SPLINE
SPL {X  -160.000, Y  +472.196, Z    +0.000, E1   +56.977, E3 +201376.828}
SPL {X  -160.000, Y  +448.172, Z    +0.000, E1   +58.434, E3 +201399.523}
SPL {X  -160.000, Y  +423.986, Z    +0.000, E1   +59.836, E3 +201420.777}
SPL {X  -160.000, Y  +398.875, Z    +0.000, E1   +61.100, E3 +201442.325}
SPL {X  -159.733, Y  +376.466, Z    +0.000, E1   +61.765, E3 +201463.514}
SPL {X  -158.128, Y  +361.299, Z    +0.000, E1   +61.520, E3 +201482.494}
SPL {X  -155.661, Y  +348.690, Z    +0.000, E1   +61.132, E3 +201499.450}
SPL {X  -152.251, Y  +336.510, Z    +0.000, E1   +60.617, E3 +201516.783}
SPL {X  -148.078, Y  +325.096, Z    +0.000, E1   +59.928, E3 +201533.911}
SPL {X  -143.290, Y  +314.510, Z    +0.000, E1   +59.129, E3 +201550.534}
SPL {X  -139.113, Y  +306.659, Z    +0.000, E1   +58.310, E3 +201563.385}
SPL {X  -135.700, Y  +300.932, Z    +0.000, E1   +57.683, E3 +201572.881}
SPL {X  -117.539, Y  +277.143, Z    +0.000, E1   +48.559, E3 +201687.567}
ENDSPLINE

SPLINE
SPL {X  -150.734, Y  +332.041, Z    +0.000, E1   +31.286, E3 +201790.232}
SPL {X  -159.235, Y  +370.077, Z    +0.000, E1   +12.240, E3 +201803.586}
SPL {X  -159.991, Y  +384.025, Z    +0.000, E1    +2.884, E3 +201805.135}
SPL {X  -160.000, Y  +388.170, Z    +0.000, E1    -0.470, E3 +201805.266}
SPL {X  -160.000, Y  +392.385, Z    +0.000, E1    -5.697, E3 +201805.456}
SPL {X  -160.000, Y  +398.918, Z    +0.000, E1   -15.420, E3 +201806.134}
SPL {X  -160.000, Y  +410.991, Z    +0.000, E1   -32.499, E3 +201808.629}
SPL {X  -160.000, Y  +455.466, Z    +0.000, E1   -56.407, E3 +201829.528}
SPL {X  -160.000, Y  +554.875, Z    +0.000, E1   -61.915, E3 +201911.432}
SPL {X  -160.000, Y  +571.700, Z    +0.000, E1   -61.918, E3 +201930.509}
SPL {X  -160.000, Y  +587.975, Z    +0.000, E1   -61.909, E3 +201948.976}
SPL {X  -160.000, Y  +604.690, Z    +0.000, E1   -61.922, E3 +201967.905}
SPL {X  -160.000, Y  +621.475, Z    +0.000, E1   -61.913, E3 +201986.957}
SPL {X  -160.000, Y  +638.005, Z    +0.000, E1   -61.917, E3 +202005.687}
SPL {X  -160.000, Y  +655.083, Z    +0.000, E1   -61.921, E3 +202025.048}
SPL {X  -160.000, Y  +671.910, Z    +0.000, E1   -61.915, E3 +202044.142}
SPL {X  -159.476, Y  +687.338, Z    +0.000, E1   -61.835, E3 +202062.194}
SPL {X  -157.928, Y  +700.064, Z    +0.000, E1   -61.593, E3 +202078.259}
SPL {X  -155.236, Y  +713.154, Z    +0.000, E1   -61.225, E3 +202095.806}
SPL {X  -151.860, Y  +724.785, Z    +0.000, E1   -60.654, E3 +202112.479}
SPL {X  -148.451, Y  +734.085, Z    +0.000, E1   -60.099, E3 +202126.404}
SPL {X  -144.033, Y  +744.073, Z    +0.000, E1   -59.381, E3 +202141.924}
SPL {X  -139.170, Y  +753.341, Z    +0.000, E1   -58.489, E3 +202156.945}
SPL {X  -135.320, Y  +759.772, Z    +0.000, E1   -57.727, E3 +202167.655}
SPL {X  -117.185, Y  +783.339, Z    +0.000, E1   -48.966, E3 +202276.041}
ENDSPLINE

SPLINE
SPL {X  -142.074, Y  +747.987, Z    +0.000, E1   -38.326, E3 +202374.735}
SPL {X  -154.075, Y  +717.539, Z    +0.000, E1   -26.988, E3 +202393.892}
SPL {X  -158.904, Y  +693.092, Z    +0.000, E1   -14.171, E3 +202400.683}
SPL {X  -159.937, Y  +678.885, Z    +0.000, E1    -4.971, E3 +202402.510}
SPL {X  -160.000, Y  +672.790, Z    +0.000, E1    -0.387, E3 +202402.778}
SPL {X  -160.000, Y  +669.961, Z    +0.000, E1    +2.696, E3 +202402.855}
SPL {X  -160.000, Y  +663.591, Z    +0.000, E1   +11.688, E3 +202403.349}
SPL {X  -160.000, Y  +654.521, Z    +0.000, E1   +25.997, E3 +202404.707}
SPL {X  -160.000, Y  +642.364, Z    +0.000, E1   +40.387, E3 +202408.009}
SPL {X  -160.000, Y  +597.330, Z    +0.000, E1   +58.145, E3 +202430.920}
SPL {X  -160.000, Y  +516.293, Z    +0.000, E1   +61.751, E3 +202497.977}
SPL {X  -160.000, Y  +506.292, Z    +0.000, E1   +61.780, E3 +202509.311}
SPL {X  -160.000, Y  +494.139, Z    +0.000, E1   +61.770, E3 +202523.182}
SPL {X  -160.000, Y  +480.560, Z    +0.000, E1   +61.503, E3 +202540.979}
ENDSPLINE

SPLINE
SPL {X  -160.000, Y  +495.136, Z    +0.000, E1   +55.416, E3 +202562.485}
ENDSPLINE

SPLINE
SPL {X  -160.000, Y  +472.196, Z    +0.000, E1   +56.977, E3 +202585.160}
SPL {X  -160.000, Y  +448.172, Z    +0.000, E1   +58.434, E3 +202607.855}
SPL {X  -160.000, Y  +423.986, Z    +0.000, E1   +59.836, E3 +202629.108}
SPL {X  -160.000, Y  +398.875, Z    +0.000, E1   +61.100, E3 +202650.656}
SPL {X  -159.733, Y  +376.466, Z    +0.000, E1   +61.765, E3 +202671.846}
SPL {X  -158.128, Y  +361.299, Z    +0.000, E1   +61.520, E3 +202690.826}
SPL {X  -155.661, Y  +348.690, Z    +0.000, E1   +61.132, E3 +202707.782}
SPL {X  -152.251, Y  +336.510, Z    +0.000, E1   +60.617, E3 +202725.114}
SPL {X  -148.078, Y  +325.096, Z    +0.000, E1   +59.928, E3 +202742.243}
SPL {X  -143.290, Y  +314.510, Z    +0.000, E1   +59.129, E3 +202758.866}
SPL {X  -139.113, Y  +306.659, Z    +0.000, E1   +58.310, E3 +202771.716}
SPL {X  -135.700, Y  +300.932, Z    +0.000, E1   +57.683, E3 +202781.213}
SPL {X  -117.539, Y  +277.143, Z    +0.000, E1   +48.559, E3 +202895.899}
ENDSPLINE

SPLINE
SPL {X  -150.734, Y  +332.041, Z    +0.000, E1   +31.286, E3 +202998.564}
SPL {X  -159.235, Y  +370.077, Z    +0.000, E1   +12.240, E3 +203011.918}
SPL {X  -159.991, Y  +384.025, Z    +0.000, E1    +2.884, E3 +203013.467}
SPL {X  -160.000, Y  +388.170, Z    +0.000, E1    -0.470, E3 +203013.597}
SPL {X  -160.000, Y  +392.385, Z    +0.000, E1    -5.697, E3 +203013.787}
SPL {X  -160.000, Y  +398.918, Z    +0.000, E1   -15.420, E3 +203014.466}
SPL {X  -160.000, Y  +410.991, Z    +0.000, E1   -32.499, E3 +203016.961}
SPL {X  -160.000, Y  +455.466, Z    +0.000, E1   -56.407, E3 +203037.860}
SPL {X  -160.000, Y  +554.875, Z    +0.000, E1   -61.915, E3 +203119.764}
SPL {X  -160.000, Y  +571.700, Z    +0.000, E1   -61.918, E3 +203138.841}
SPL {X  -160.000, Y  +587.975, Z    +0.000, E1   -61.909, E3 +203157.307}
SPL {X  -160.000, Y  +604.690, Z    +0.000, E1   -61.922, E3 +203176.237}
SPL {X  -160.000, Y  +621.475, Z    +0.000, E1   -61.913, E3 +203195.288}
SPL {X  -160.000, Y  +638.005, Z    +0.000, E1   -61.917, E3 +203214.019}
SPL {X  -160.000, Y  +655.083, Z    +0.000, E1   -61.921, E3 +203233.380}
SPL {X  -160.000, Y  +671.910, Z    +0.000, E1   -61.915, E3 +203252.474}
SPL {X  -159.476, Y  +687.338, Z    +0.000, E1   -61.835, E3 +203270.526}
SPL {X  -157.928, Y  +700.064, Z    +0.000, E1   -61.593, E3 +203286.591}
SPL {X  -155.236, Y  +713.154, Z    +0.000, E1   -61.225, E3 +203304.138}
SPL {X  -151.860, Y  +724.785, Z    +0.000, E1   -60.654, E3 +203320.810}
SPL {X  -148.451, Y  +734.085, Z    +0.000, E1   -60.099, E3 +203334.735}
SPL {X  -144.033, Y  +744.073, Z    +0.000, E1   -59.381, E3 +203350.256}
SPL {X  -139.170, Y  +753.341, Z    +0.000, E1   -58.489, E3 +203365.277}
SPL {X  -135.320, Y  +759.772, Z    +0.000, E1   -57.727, E3 +203375.987}
SPL {X  -117.185, Y  +783.339, Z    +0.000, E1   -48.966, E3 +203484.373}
ENDSPLINE

SPLINE
SPL {X  -142.074, Y  +747.987, Z    +0.000, E1   -38.326, E3 +203583.067}
SPL {X  -154.075, Y  +717.539, Z    +0.000, E1   -26.988, E3 +203602.224}
SPL {X  -158.904, Y  +693.092, Z    +0.000, E1   -14.171, E3 +203609.015}
SPL {X  -159.937, Y  +678.885, Z    +0.000, E1    -4.971, E3 +203610.842}
SPL {X  -160.000, Y  +672.790, Z    +0.000, E1    -0.387, E3 +203611.110}
SPL {X  -160.000, Y  +669.961, Z    +0.000, E1    +2.696, E3 +203611.187}
SPL {X  -160.000, Y  +663.591, Z    +0.000, E1   +11.688, E3 +203611.681}
SPL {X  -160.000, Y  +654.521, Z    +0.000, E1   +25.997, E3 +203613.039}
SPL {X  -160.000, Y  +642.364, Z    +0.000, E1   +40.387, E3 +203616.341}
SPL {X  -160.000, Y  +597.330, Z    +0.000, E1   +58.145, E3 +203639.252}
SPL {X  -160.000, Y  +507.195, Z    +0.000, E1   +61.792, E3 +203716.583}
SPL {X  -160.000, Y  +494.139, Z    +0.000, E1   +61.770, E3 +203731.513}
SPL {X  -160.000, Y  +480.560, Z    +0.000, E1   +61.503, E3 +203749.310}
ENDSPLINE

SPLINE
SPL {X  -160.000, Y  +495.136, Z    +0.000, E1   +55.416, E3 +203770.817}
ENDSPLINE

SPLINE
SPL {X  -160.000, Y  +472.196, Z    +0.000, E1   +56.977, E3 +203793.492}
SPL {X  -160.000, Y  +448.172, Z    +0.000, E1   +58.434, E3 +203816.187}
SPL {X  -160.000, Y  +423.986, Z    +0.000, E1   +59.836, E3 +203837.440}
SPL {X  -160.000, Y  +398.875, Z    +0.000, E1   +61.100, E3 +203858.988}
SPL {X  -159.733, Y  +376.466, Z    +0.000, E1   +61.765, E3 +203880.178}
SPL {X  -158.128, Y  +361.299, Z    +0.000, E1   +61.520, E3 +203899.157}
SPL {X  -155.661, Y  +348.690, Z    +0.000, E1   +61.132, E3 +203916.113}
SPL {X  -152.251, Y  +336.510, Z    +0.000, E1   +60.617, E3 +203933.446}
SPL {X  -148.078, Y  +325.096, Z    +0.000, E1   +59.928, E3 +203950.575}
SPL {X  -143.290, Y  +314.510, Z    +0.000, E1   +59.129, E3 +203967.198}
SPL {X  -139.113, Y  +306.659, Z    +0.000, E1   +58.310, E3 +203980.048}
SPL {X  -135.700, Y  +300.932, Z    +0.000, E1   +57.683, E3 +203989.545}
SPL {X  -117.539, Y  +277.143, Z    +0.000, E1   +48.559, E3 +204104.231}
ENDSPLINE

SPLINE
SPL {X  -150.734, Y  +332.041, Z    +0.000, E1   +31.286, E3 +204206.896}
SPL {X  -159.235, Y  +370.077, Z    +0.000, E1   +12.240, E3 +204220.250}
SPL {X  -159.991, Y  +384.025, Z    +0.000, E1    +2.884, E3 +204221.798}
SPL {X  -160.000, Y  +388.170, Z    +0.000, E1    -0.470, E3 +204221.929}
SPL {X  -160.000, Y  +392.385, Z    +0.000, E1    -5.697, E3 +204222.119}
SPL {X  -160.000, Y  +398.918, Z    +0.000, E1   -15.420, E3 +204222.798}
SPL {X  -160.000, Y  +410.991, Z    +0.000, E1   -32.499, E3 +204225.293}
SPL {X  -160.000, Y  +455.466, Z    +0.000, E1   -56.407, E3 +204246.192}
SPL {X  -160.000, Y  +554.875, Z    +0.000, E1   -61.915, E3 +204328.096}
SPL {X  -160.000, Y  +571.700, Z    +0.000, E1   -61.918, E3 +204347.173}
SPL {X  -160.000, Y  +587.975, Z    +0.000, E1   -61.909, E3 +204365.639}
SPL {X  -160.000, Y  +604.690, Z    +0.000, E1   -61.922, E3 +204384.568}
SPL {X  -160.000, Y  +621.475, Z    +0.000, E1   -61.913, E3 +204403.620}
SPL {X  -160.000, Y  +638.005, Z    +0.000, E1   -61.917, E3 +204422.351}
SPL {X  -160.000, Y  +655.083, Z    +0.000, E1   -61.921, E3 +204441.712}
SPL {X  -160.000, Y  +671.910, Z    +0.000, E1   -61.915, E3 +204460.806}
SPL {X  -159.476, Y  +687.338, Z    +0.000, E1   -61.835, E3 +204478.858}
SPL {X  -157.928, Y  +700.064, Z    +0.000, E1   -61.593, E3 +204494.922}
SPL {X  -155.236, Y  +713.154, Z    +0.000, E1   -61.225, E3 +204512.469}
SPL {X  -151.860, Y  +724.785, Z    +0.000, E1   -60.654, E3 +204529.142}
SPL {X  -148.451, Y  +734.085, Z    +0.000, E1   -60.099, E3 +204543.067}
SPL {X  -144.033, Y  +744.073, Z    +0.000, E1   -59.381, E3 +204558.587}
SPL {X  -139.170, Y  +753.341, Z    +0.000, E1   -58.489, E3 +204573.609}
SPL {X  -135.320, Y  +759.772, Z    +0.000, E1   -57.727, E3 +204584.319}
SPL {X  -117.185, Y  +783.339, Z    +0.000, E1   -48.966, E3 +204692.705}
ENDSPLINE

SPLINE
SPL {X  -142.074, Y  +747.987, Z    +0.000, E1   -38.326, E3 +204791.398}
SPL {X  -154.075, Y  +717.539, Z    +0.000, E1   -26.988, E3 +204810.555}
SPL {X  -158.904, Y  +693.092, Z    +0.000, E1   -14.171, E3 +204817.346}
SPL {X  -159.937, Y  +678.885, Z    +0.000, E1    -4.971, E3 +204819.174}
SPL {X  -160.000, Y  +672.790, Z    +0.000, E1    -0.387, E3 +204819.442}
SPL {X  -160.000, Y  +669.961, Z    +0.000, E1    +2.696, E3 +204819.518}
SPL {X  -160.000, Y  +663.591, Z    +0.000, E1   +11.688, E3 +204820.013}
SPL {X  -160.000, Y  +654.521, Z    +0.000, E1   +25.997, E3 +204821.370}
SPL {X  -160.000, Y  +642.364, Z    +0.000, E1   +40.387, E3 +204824.673}
SPL {X  -160.000, Y  +597.330, Z    +0.000, E1   +58.145, E3 +204847.584}
SPL {X  -160.000, Y  +507.195, Z    +0.000, E1   +61.792, E3 +204924.915}
SPL {X  -160.000, Y  +494.139, Z    +0.000, E1   +61.770, E3 +204939.845}
SPL {X  -160.000, Y  +480.560, Z    +0.000, E1   +61.503, E3 +204957.642}
ENDSPLINE

SPLINE
SPL {X  -160.000, Y  +495.136, Z    +0.000, E1   +55.416, E3 +204979.149}
ENDSPLINE

SPLINE
SPL {X  -160.000, Y  +472.196, Z    +0.000, E1   +56.977, E3 +205001.824}
SPL {X  -160.000, Y  +448.172, Z    +0.000, E1   +58.434, E3 +205024.518}
SPL {X  -160.000, Y  +423.986, Z    +0.000, E1   +59.836, E3 +205045.772}
SPL {X  -160.000, Y  +398.875, Z    +0.000, E1   +61.100, E3 +205067.320}
SPL {X  -159.733, Y  +376.466, Z    +0.000, E1   +61.765, E3 +205088.509}
SPL {X  -158.128, Y  +361.299, Z    +0.000, E1   +61.520, E3 +205107.489}
SPL {X  -155.661, Y  +348.690, Z    +0.000, E1   +61.132, E3 +205124.445}
SPL {X  -152.251, Y  +336.510, Z    +0.000, E1   +60.617, E3 +205141.778}
SPL {X  -148.078, Y  +325.096, Z    +0.000, E1   +59.928, E3 +205158.906}
SPL {X  -143.290, Y  +314.510, Z    +0.000, E1   +59.129, E3 +205175.529}
SPL {X  -139.113, Y  +306.659, Z    +0.000, E1   +58.310, E3 +205188.380}
SPL {X  -135.700, Y  +300.932, Z    +0.000, E1   +57.683, E3 +205197.877}
SPL {X  -117.539, Y  +277.143, Z    +0.000, E1   +48.559, E3 +205312.563}
ENDSPLINE

SPLINE
SPL {X  -150.734, Y  +332.041, Z    +0.000, E1   +31.286, E3 +205415.227}
SPL {X  -159.235, Y  +370.077, Z    +0.000, E1   +12.240, E3 +205428.581}
SPL {X  -159.991, Y  +384.025, Z    +0.000, E1    +2.884, E3 +205430.130}
SPL {X  -160.000, Y  +388.170, Z    +0.000, E1    -0.470, E3 +205430.261}
SPL {X  -160.000, Y  +392.385, Z    +0.000, E1    -5.697, E3 +205430.451}
SPL {X  -160.000, Y  +398.918, Z    +0.000, E1   -15.420, E3 +205431.130}
SPL {X  -160.000, Y  +410.991, Z    +0.000, E1   -32.499, E3 +205433.625}
SPL {X  -160.000, Y  +455.466, Z    +0.000, E1   -56.407, E3 +205454.524}
SPL {X  -160.000, Y  +554.875, Z    +0.000, E1   -61.915, E3 +205536.427}
SPL {X  -160.000, Y  +571.700, Z    +0.000, E1   -61.918, E3 +205555.504}
SPL {X  -160.000, Y  +587.975, Z    +0.000, E1   -61.909, E3 +205573.971}
SPL {X  -160.000, Y  +604.690, Z    +0.000, E1   -61.922, E3 +205592.900}
SPL {X  -160.000, Y  +621.475, Z    +0.000, E1   -61.913, E3 +205611.952}
SPL {X  -160.000, Y  +638.005, Z    +0.000, E1   -61.917, E3 +205630.682}
SPL {X  -160.000, Y  +655.083, Z    +0.000, E1   -61.921, E3 +205650.044}
SPL {X  -160.000, Y  +671.910, Z    +0.000, E1   -61.915, E3 +205669.138}
SPL {X  -159.476, Y  +687.338, Z    +0.000, E1   -61.835, E3 +205687.190}
SPL {X  -157.928, Y  +700.064, Z    +0.000, E1   -61.593, E3 +205703.254}
SPL {X  -155.236, Y  +713.154, Z    +0.000, E1   -61.225, E3 +205720.801}
SPL {X  -151.860, Y  +724.785, Z    +0.000, E1   -60.654, E3 +205737.474}
SPL {X  -148.451, Y  +734.085, Z    +0.000, E1   -60.099, E3 +205751.399}
SPL {X  -144.033, Y  +744.073, Z    +0.000, E1   -59.381, E3 +205766.919}
SPL {X  -139.170, Y  +753.341, Z    +0.000, E1   -58.489, E3 +205781.941}
SPL {X  -135.320, Y  +759.772, Z    +0.000, E1   -57.727, E3 +205792.650}
SPL {X  -117.185, Y  +783.339, Z    +0.000, E1   -48.966, E3 +205901.037}
ENDSPLINE

SPLINE
SPL {X  -142.074, Y  +747.987, Z    +0.000, E1   -38.326, E3 +205999.730}
SPL {X  -154.075, Y  +717.539, Z    +0.000, E1   -26.988, E3 +206018.887}
SPL {X  -158.904, Y  +693.092, Z    +0.000, E1   -14.171, E3 +206025.678}
SPL {X  -159.937, Y  +678.885, Z    +0.000, E1    -4.971, E3 +206027.505}
SPL {X  -160.000, Y  +672.790, Z    +0.000, E1    -0.387, E3 +206027.773}
SPL {X  -160.000, Y  +669.961, Z    +0.000, E1    +2.696, E3 +206027.850}
SPL {X  -160.000, Y  +663.591, Z    +0.000, E1   +11.688, E3 +206028.344}
SPL {X  -160.000, Y  +654.521, Z    +0.000, E1   +25.997, E3 +206029.702}
SPL {X  -160.000, Y  +642.364, Z    +0.000, E1   +40.387, E3 +206033.004}
SPL {X  -160.000, Y  +597.330, Z    +0.000, E1   +58.145, E3 +206055.915}
SPL {X  -160.000, Y  +516.293, Z    +0.000, E1   +61.751, E3 +206122.973}
SPL {X  -160.000, Y  +506.292, Z    +0.000, E1   +61.780, E3 +206134.306}
SPL {X  -160.000, Y  +494.139, Z    +0.000, E1   +61.770, E3 +206148.177}
SPL {X  -160.000, Y  +480.560, Z    +0.000, E1   +61.503, E3 +206165.974}
ENDSPLINE

SPLINE
SPL {X  -160.000, Y  +495.136, Z    +0.000, E1   +55.416, E3 +206187.480}
ENDSPLINE

SPLINE
SPL {X  -160.000, Y  +472.196, Z    +0.000, E1   +56.977, E3 +206210.155}
SPL {X  -160.000, Y  +448.172, Z    +0.000, E1   +58.434, E3 +206232.850}
SPL {X  -160.000, Y  +423.986, Z    +0.000, E1   +59.836, E3 +206254.104}
SPL {X  -160.000, Y  +398.875, Z    +0.000, E1   +61.100, E3 +206275.652}
SPL {X  -159.733, Y  +376.466, Z    +0.000, E1   +61.765, E3 +206296.841}
SPL {X  -158.128, Y  +361.299, Z    +0.000, E1   +61.520, E3 +206315.821}
SPL {X  -155.661, Y  +348.690, Z    +0.000, E1   +61.132, E3 +206332.777}
SPL {X  -152.251, Y  +336.510, Z    +0.000, E1   +60.617, E3 +206350.110}
SPL {X  -148.078, Y  +325.096, Z    +0.000, E1   +59.928, E3 +206367.238}
SPL {X  -143.290, Y  +314.510, Z    +0.000, E1   +59.129, E3 +206383.861}
SPL {X  -139.113, Y  +306.659, Z    +0.000, E1   +58.310, E3 +206396.712}
SPL {X  -135.700, Y  +300.932, Z    +0.000, E1   +57.683, E3 +206406.208}
SPL {X  -117.539, Y  +277.143, Z    +0.000, E1   +48.559, E3 +206520.894}
ENDSPLINE

SPLINE
SPL {X  -150.734, Y  +332.041, Z    +0.000, E1   +31.286, E3 +206623.559}
SPL {X  -159.235, Y  +370.077, Z    +0.000, E1   +12.240, E3 +206636.913}
SPL {X  -159.991, Y  +384.025, Z    +0.000, E1    +2.884, E3 +206638.462}
SPL {X  -160.000, Y  +388.170, Z    +0.000, E1    -0.470, E3 +206638.593}
SPL {X  -160.000, Y  +392.385, Z    +0.000, E1    -5.697, E3 +206638.783}
SPL {X  -160.000, Y  +398.918, Z    +0.000, E1   -15.420, E3 +206639.461}
SPL {X  -160.000, Y  +410.991, Z    +0.000, E1   -32.499, E3 +206641.956}
SPL {X  -160.000, Y  +455.466, Z    +0.000, E1   -56.407, E3 +206662.855}
SPL {X  -160.000, Y  +554.875, Z    +0.000, E1   -61.915, E3 +206744.759}
SPL {X  -160.000, Y  +571.700, Z    +0.000, E1   -61.918, E3 +206763.836}
SPL {X  -160.000, Y  +587.975, Z    +0.000, E1   -61.909, E3 +206782.303}
SPL {X  -160.000, Y  +604.690, Z    +0.000, E1   -61.922, E3 +206801.232}
SPL {X  -160.000, Y  +621.475, Z    +0.000, E1   -61.913, E3 +206820.284}
SPL {X  -160.000, Y  +638.005, Z    +0.000, E1   -61.917, E3 +206839.014}
SPL {X  -160.000, Y  +655.083, Z    +0.000, E1   -61.921, E3 +206858.375}
SPL {X  -160.000, Y  +671.910, Z    +0.000, E1   -61.915, E3 +206877.469}
SPL {X  -159.476, Y  +687.338, Z    +0.000, E1   -61.835, E3 +206895.521}
SPL {X  -157.928, Y  +700.064, Z    +0.000, E1   -61.593, E3 +206911.586}
SPL {X  -155.236, Y  +713.154, Z    +0.000, E1   -61.225, E3 +206929.133}
SPL {X  -151.860, Y  +724.785, Z    +0.000, E1   -60.654, E3 +206945.806}
SPL {X  -148.451, Y  +734.085, Z    +0.000, E1   -60.099, E3 +206959.731}
SPL {X  -144.033, Y  +744.073, Z    +0.000, E1   -59.381, E3 +206975.251}
SPL {X  -139.170, Y  +753.341, Z    +0.000, E1   -58.489, E3 +206990.273}
SPL {X  -135.320, Y  +759.772, Z    +0.000, E1   -57.727, E3 +207000.982}
SPL {X  -117.185, Y  +783.339, Z    +0.000, E1   -48.966, E3 +207109.368}
ENDSPLINE

SPLINE
SPL {X  -142.074, Y  +747.987, Z    +0.000, E1   -38.326, E3 +207208.062}
SPL {X  -154.075, Y  +717.539, Z    +0.000, E1   -26.988, E3 +207227.219}
SPL {X  -158.904, Y  +693.092, Z    +0.000, E1   -14.171, E3 +207234.010}
SPL {X  -159.937, Y  +678.885, Z    +0.000, E1    -4.971, E3 +207235.837}
SPL {X  -160.000, Y  +672.790, Z    +0.000, E1    -0.387, E3 +207236.105}
SPL {X  -160.000, Y  +669.961, Z    +0.000, E1    +2.696, E3 +207236.182}
SPL {X  -160.000, Y  +663.591, Z    +0.000, E1   +11.688, E3 +207236.676}
SPL {X  -160.000, Y  +654.521, Z    +0.000, E1   +25.997, E3 +207238.034}
SPL {X  -160.000, Y  +642.364, Z    +0.000, E1   +40.387, E3 +207241.336}
SPL {X  -160.000, Y  +597.330, Z    +0.000, E1   +58.145, E3 +207264.247}
SPL {X  -160.000, Y  +507.195, Z    +0.000, E1   +61.792, E3 +207341.578}
SPL {X  -160.000, Y  +494.139, Z    +0.000, E1   +61.770, E3 +207356.509}
SPL {X  -160.000, Y  +480.560, Z    +0.000, E1   +61.503, E3 +207374.306}
ENDSPLINE

SPLINE
SPL {X  -160.000, Y  +495.136, Z    +0.000, E1   +55.416, E3 +207395.812}
ENDSPLINE

SPLINE
SPL {X  -160.000, Y  +472.196, Z    +0.000, E1   +56.977, E3 +207418.487}
SPL {X  -160.000, Y  +448.172, Z    +0.000, E1   +58.434, E3 +207441.182}
SPL {X  -160.000, Y  +423.986, Z    +0.000, E1   +59.836, E3 +207462.435}
SPL {X  -160.000, Y  +398.875, Z    +0.000, E1   +61.100, E3 +207483.983}
SPL {X  -159.733, Y  +376.466, Z    +0.000, E1   +61.765, E3 +207505.173}
SPL {X  -158.128, Y  +361.299, Z    +0.000, E1   +61.520, E3 +207524.153}
SPL {X  -155.661, Y  +348.690, Z    +0.000, E1   +61.132, E3 +207541.109}
SPL {X  -152.251, Y  +336.510, Z    +0.000, E1   +60.617, E3 +207558.441}
SPL {X  -148.078, Y  +325.096, Z    +0.000, E1   +59.928, E3 +207575.570}
SPL {X  -143.290, Y  +314.510, Z    +0.000, E1   +59.129, E3 +207592.193}
SPL {X  -139.113, Y  +306.659, Z    +0.000, E1   +58.310, E3 +207605.043}
SPL {X  -135.700, Y  +300.932, Z    +0.000, E1   +57.683, E3 +207614.540}
SPL {X  -117.539, Y  +277.143, Z    +0.000, E1   +48.559, E3 +207729.226}
ENDSPLINE

SPLINE
SPL {X  -150.734, Y  +332.041, Z    +0.000, E1   +31.286, E3 +207831.891}
SPL {X  -159.235, Y  +370.077, Z    +0.000, E1   +12.240, E3 +207845.245}
SPL {X  -159.991, Y  +384.025, Z    +0.000, E1    +2.884, E3 +207846.794}
SPL {X  -160.000, Y  +388.170, Z    +0.000, E1    -0.470, E3 +207846.924}
SPL {X  -160.000, Y  +392.385, Z    +0.000, E1    -5.697, E3 +207847.114}
SPL {X  -160.000, Y  +398.918, Z    +0.000, E1   -15.420, E3 +207847.793}
SPL {X  -160.000, Y  +410.991, Z    +0.000, E1   -32.499, E3 +207850.288}
SPL {X  -160.000, Y  +455.466, Z    +0.000, E1   -56.407, E3 +207871.187}
SPL {X  -160.000, Y  +554.875, Z    +0.000, E1   -61.915, E3 +207953.091}
SPL {X  -160.000, Y  +571.700, Z    +0.000, E1   -61.918, E3 +207972.168}
SPL {X  -160.000, Y  +587.975, Z    +0.000, E1   -61.909, E3 +207990.634}
SPL {X  -160.000, Y  +604.690, Z    +0.000, E1   -61.922, E3 +208009.564}
SPL {X  -160.000, Y  +621.475, Z    +0.000, E1   -61.913, E3 +208028.615}
SPL {X  -160.000, Y  +638.005, Z    +0.000, E1   -61.917, E3 +208047.346}
SPL {X  -160.000, Y  +655.083, Z    +0.000, E1   -61.921, E3 +208066.707}
SPL {X  -160.000, Y  +671.910, Z    +0.000, E1   -61.915, E3 +208085.801}
SPL {X  -159.476, Y  +687.338, Z    +0.000, E1   -61.835, E3 +208103.853}
SPL {X  -157.928, Y  +700.064, Z    +0.000, E1   -61.593, E3 +208119.918}
SPL {X  -155.236, Y  +713.154, Z    +0.000, E1   -61.225, E3 +208137.465}
SPL {X  -151.860, Y  +724.785, Z    +0.000, E1   -60.654, E3 +208154.137}
SPL {X  -148.451, Y  +734.085, Z    +0.000, E1   -60.099, E3 +208168.062}
SPL {X  -144.033, Y  +744.073, Z    +0.000, E1   -59.381, E3 +208183.583}
SPL {X  -139.170, Y  +753.341, Z    +0.000, E1   -58.489, E3 +208198.604}
SPL {X  -135.320, Y  +759.772, Z    +0.000, E1   -57.727, E3 +208209.314}
SPL {X  -117.185, Y  +783.339, Z    +0.000, E1   -48.966, E3 +208317.700}
ENDSPLINE

SPLINE
SPL {X  -142.074, Y  +747.987, Z    +0.000, E1   -38.326, E3 +208416.394}
SPL {X  -154.075, Y  +717.539, Z    +0.000, E1   -26.988, E3 +208435.551}
SPL {X  -158.904, Y  +693.092, Z    +0.000, E1   -14.171, E3 +208442.342}
SPL {X  -159.937, Y  +678.885, Z    +0.000, E1    -4.971, E3 +208444.169}
SPL {X  -160.000, Y  +672.790, Z    +0.000, E1    -0.387, E3 +208444.437}
SPL {X  -160.000, Y  +669.961, Z    +0.000, E1    +2.696, E3 +208444.514}
SPL {X  -160.000, Y  +663.591, Z    +0.000, E1   +11.688, E3 +208445.008}
SPL {X  -160.000, Y  +654.521, Z    +0.000, E1   +25.997, E3 +208446.366}
SPL {X  -160.000, Y  +642.364, Z    +0.000, E1   +40.387, E3 +208449.668}
SPL {X  -160.000, Y  +597.330, Z    +0.000, E1   +58.145, E3 +208472.579}
SPL {X  -160.000, Y  +507.195, Z    +0.000, E1   +61.792, E3 +208549.910}
SPL {X  -160.000, Y  +494.139, Z    +0.000, E1   +61.770, E3 +208564.840}
SPL {X  -160.000, Y  +480.560, Z    +0.000, E1   +61.503, E3 +208582.637}
ENDSPLINE

SPLINE
SPL {X  -160.000, Y  +495.136, Z    +0.000, E1   +55.416, E3 +208604.144}
ENDSPLINE

SPLINE
SPL {X  -160.000, Y  +472.196, Z    +0.000, E1   +56.977, E3 +208626.819}
SPL {X  -160.000, Y  +448.172, Z    +0.000, E1   +58.434, E3 +208649.514}
SPL {X  -160.000, Y  +423.986, Z    +0.000, E1   +59.836, E3 +208670.767}
SPL {X  -160.000, Y  +398.875, Z    +0.000, E1   +61.100, E3 +208692.315}
SPL {X  -159.733, Y  +376.466, Z    +0.000, E1   +61.765, E3 +208713.505}
SPL {X  -158.128, Y  +361.299, Z    +0.000, E1   +61.520, E3 +208732.484}
SPL {X  -155.661, Y  +348.690, Z    +0.000, E1   +61.132, E3 +208749.440}
SPL {X  -152.251, Y  +336.510, Z    +0.000, E1   +60.617, E3 +208766.773}
SPL {X  -148.078, Y  +325.096, Z    +0.000, E1   +59.928, E3 +208783.902}
SPL {X  -143.290, Y  +314.510, Z    +0.000, E1   +59.129, E3 +208800.525}
SPL {X  -139.113, Y  +306.659, Z    +0.000, E1   +58.310, E3 +208813.375}
SPL {X  -135.700, Y  +300.932, Z    +0.000, E1   +57.683, E3 +208822.872}
SPL {X  -117.539, Y  +277.143, Z    +0.000, E1   +48.559, E3 +208937.558}
ENDSPLINE

SPLINE
SPL {X  -150.734, Y  +332.041, Z    +0.000, E1   +31.286, E3 +209040.223}
SPL {X  -159.235, Y  +370.077, Z    +0.000, E1   +12.240, E3 +209053.577}
SPL {X  -159.991, Y  +384.025, Z    +0.000, E1    +2.884, E3 +209055.125}
SPL {X  -160.000, Y  +388.170, Z    +0.000, E1    -0.470, E3 +209055.256}
SPL {X  -160.000, Y  +392.385, Z    +0.000, E1    -5.697, E3 +209055.446}
SPL {X  -160.000, Y  +398.918, Z    +0.000, E1   -15.420, E3 +209056.125}
SPL {X  -160.000, Y  +410.991, Z    +0.000, E1   -32.499, E3 +209058.620}
SPL {X  -160.000, Y  +455.466, Z    +0.000, E1   -56.407, E3 +209079.519}
SPL {X  -160.000, Y  +554.875, Z    +0.000, E1   -61.915, E3 +209161.423}
SPL {X  -160.000, Y  +571.700, Z    +0.000, E1   -61.918, E3 +209180.500}
SPL {X  -160.000, Y  +587.975, Z    +0.000, E1   -61.909, E3 +209198.966}
SPL {X  -160.000, Y  +604.690, Z    +0.000, E1   -61.922, E3 +209217.895}
SPL {X  -160.000, Y  +621.475, Z    +0.000, E1   -61.913, E3 +209236.947}
SPL {X  -160.000, Y  +638.005, Z    +0.000, E1   -61.917, E3 +209255.678}
SPL {X  -160.000, Y  +655.083, Z    +0.000, E1   -61.921, E3 +209275.039}
SPL {X  -160.000, Y  +671.910, Z    +0.000, E1   -61.915, E3 +209294.133}
SPL {X  -159.476, Y  +687.338, Z    +0.000, E1   -61.835, E3 +209312.185}
SPL {X  -157.928, Y  +700.064, Z    +0.000, E1   -61.593, E3 +209328.249}
SPL {X  -155.236, Y  +713.154, Z    +0.000, E1   -61.225, E3 +209345.797}
SPL {X  -151.860, Y  +724.785, Z    +0.000, E1   -60.654, E3 +209362.469}
SPL {X  -148.451, Y  +734.085, Z    +0.000, E1   -60.099, E3 +209376.394}
SPL {X  -144.033, Y  +744.073, Z    +0.000, E1   -59.381, E3 +209391.914}
SPL {X  -139.170, Y  +753.341, Z    +0.000, E1   -58.489, E3 +209406.936}
SPL {X  -135.320, Y  +759.772, Z    +0.000, E1   -57.727, E3 +209417.646}
SPL {X  -117.185, Y  +783.339, Z    +0.000, E1   -48.966, E3 +209526.032}
ENDSPLINE

SPLINE
SPL {X  -142.074, Y  +747.987, Z    +0.000, E1   -38.326, E3 +209624.725}
SPL {X  -154.075, Y  +717.539, Z    +0.000, E1   -26.988, E3 +209643.882}
SPL {X  -158.904, Y  +693.092, Z    +0.000, E1   -14.171, E3 +209650.673}
SPL {X  -159.937, Y  +678.885, Z    +0.000, E1    -4.971, E3 +209652.501}
SPL {X  -160.000, Y  +672.790, Z    +0.000, E1    -0.387, E3 +209652.769}
SPL {X  -160.000, Y  +669.961, Z    +0.000, E1    +2.696, E3 +209652.845}
SPL {X  -160.000, Y  +663.591, Z    +0.000, E1   +11.688, E3 +209653.340}
SPL {X  -160.000, Y  +654.521, Z    +0.000, E1   +25.997, E3 +209654.698}
SPL {X  -160.000, Y  +642.364, Z    +0.000, E1   +40.387, E3 +209658.000}
SPL {X  -160.000, Y  +597.330, Z    +0.000, E1   +58.145, E3 +209680.911}
SPL {X  -160.000, Y  +507.195, Z    +0.000, E1   +61.792, E3 +209758.242}
SPL {X  -160.000, Y  +494.139, Z    +0.000, E1   +61.770, E3 +209773.172}
SPL {X  -160.000, Y  +480.560, Z    +0.000, E1   +61.503, E3 +209790.969}
ENDSPLINE

SPLINE
SPL {X  -160.000, Y  +495.136, Z    +0.000, E1   +55.416, E3 +209812.476}
ENDSPLINE

SPLINE
SPL {X  -160.000, Y  +472.196, Z    +0.000, E1   +56.977, E3 +209835.151}
SPL {X  -160.000, Y  +448.172, Z    +0.000, E1   +58.434, E3 +209857.845}
SPL {X  -160.000, Y  +423.986, Z    +0.000, E1   +59.836, E3 +209879.099}
SPL {X  -160.000, Y  +398.875, Z    +0.000, E1   +61.100, E3 +209900.647}
SPL {X  -159.733, Y  +376.466, Z    +0.000, E1   +61.765, E3 +209921.837}
SPL {X  -158.128, Y  +361.299, Z    +0.000, E1   +61.520, E3 +209940.816}
SPL {X  -155.661, Y  +348.690, Z    +0.000, E1   +61.132, E3 +209957.772}
SPL {X  -152.251, Y  +336.510, Z    +0.000, E1   +60.617, E3 +209975.105}
SPL {X  -148.078, Y  +325.096, Z    +0.000, E1   +59.928, E3 +209992.233}
SPL {X  -143.290, Y  +314.510, Z    +0.000, E1   +59.129, E3 +210008.856}
SPL {X  -139.113, Y  +306.659, Z    +0.000, E1   +58.310, E3 +210021.707}
SPL {X  -135.700, Y  +300.932, Z    +0.000, E1   +57.683, E3 +210031.204}
SPL {X  -117.539, Y  +277.143, Z    +0.000, E1   +48.559, E3 +210145.890}
ENDSPLINE

SPLINE
SPL {X  -150.734, Y  +332.041, Z    +0.000, E1   +31.286, E3 +210248.554}
SPL {X  -159.235, Y  +370.077, Z    +0.000, E1   +12.240, E3 +210261.909}
SPL {X  -159.991, Y  +384.025, Z    +0.000, E1    +2.884, E3 +210263.457}
SPL {X  -160.000, Y  +388.170, Z    +0.000, E1    -0.470, E3 +210263.588}
SPL {X  -160.000, Y  +392.385, Z    +0.000, E1    -5.697, E3 +210263.778}
SPL {X  -160.000, Y  +398.918, Z    +0.000, E1   -15.420, E3 +210264.457}
SPL {X  -160.000, Y  +410.991, Z    +0.000, E1   -32.499, E3 +210266.952}
SPL {X  -160.000, Y  +455.466, Z    +0.000, E1   -56.407, E3 +210287.851}
SPL {X  -160.000, Y  +554.875, Z    +0.000, E1   -61.915, E3 +210369.754}
SPL {X  -160.000, Y  +571.700, Z    +0.000, E1   -61.918, E3 +210388.831}
SPL {X  -160.000, Y  +587.975, Z    +0.000, E1   -61.909, E3 +210407.298}
SPL {X  -160.000, Y  +604.690, Z    +0.000, E1   -61.922, E3 +210426.227}
SPL {X  -160.000, Y  +621.475, Z    +0.000, E1   -61.913, E3 +210445.279}
SPL {X  -160.000, Y  +638.005, Z    +0.000, E1   -61.917, E3 +210464.009}
SPL {X  -160.000, Y  +655.083, Z    +0.000, E1   -61.921, E3 +210483.371}
SPL {X  -160.000, Y  +671.910, Z    +0.000, E1   -61.915, E3 +210502.465}
SPL {X  -159.476, Y  +687.338, Z    +0.000, E1   -61.835, E3 +210520.517}
SPL {X  -157.928, Y  +700.064, Z    +0.000, E1   -61.593, E3 +210536.581}
SPL {X  -155.236, Y  +713.154, Z    +0.000, E1   -61.225, E3 +210554.128}
SPL {X  -151.860, Y  +724.785, Z    +0.000, E1   -60.654, E3 +210570.801}
SPL {X  -148.451, Y  +734.085, Z    +0.000, E1   -60.099, E3 +210584.726}
SPL {X  -144.033, Y  +744.073, Z    +0.000, E1   -59.381, E3 +210600.246}
SPL {X  -139.170, Y  +753.341, Z    +0.000, E1   -58.489, E3 +210615.268}
SPL {X  -135.320, Y  +759.772, Z    +0.000, E1   -57.727, E3 +210625.977}
SPL {X  -117.185, Y  +783.339, Z    +0.000, E1   -48.966, E3 +210734.364}
ENDSPLINE

SPLINE
SPL {X  -142.074, Y  +747.987, Z    +0.000, E1   -38.326, E3 +210833.057}
SPL {X  -154.075, Y  +717.539, Z    +0.000, E1   -26.988, E3 +210852.214}
SPL {X  -158.904, Y  +693.092, Z    +0.000, E1   -14.171, E3 +210859.005}
SPL {X  -159.937, Y  +678.885, Z    +0.000, E1    -4.971, E3 +210860.833}
SPL {X  -160.000, Y  +672.790, Z    +0.000, E1    -0.387, E3 +210861.100}
SPL {X  -160.000, Y  +669.961, Z    +0.000, E1    +2.696, E3 +210861.177}
SPL {X  -160.000, Y  +663.591, Z    +0.000, E1   +11.688, E3 +210861.671}
SPL {X  -160.000, Y  +654.521, Z    +0.000, E1   +25.997, E3 +210863.029}
SPL {X  -160.000, Y  +642.364, Z    +0.000, E1   +40.387, E3 +210866.331}
SPL {X  -160.000, Y  +597.330, Z    +0.000, E1   +58.145, E3 +210889.242}
SPL {X  -160.000, Y  +516.293, Z    +0.000, E1   +61.751, E3 +210956.300}
SPL {X  -160.000, Y  +506.292, Z    +0.000, E1   +61.780, E3 +210967.634}
SPL {X  -160.000, Y  +494.139, Z    +0.000, E1   +61.770, E3 +210981.504}
SPL {X  -160.000, Y  +480.560, Z    +0.000, E1   +61.503, E3 +210999.301}
ENDSPLINE

SPLINE
SPL {X  -160.000, Y  +495.136, Z    +0.000, E1   +55.416, E3 +211020.808}
ENDSPLINE

SPLINE
SPL {X  -160.000, Y  +472.196, Z    +0.000, E1   +56.977, E3 +211043.482}
SPL {X  -160.000, Y  +448.172, Z    +0.000, E1   +58.434, E3 +211066.177}
SPL {X  -160.000, Y  +423.986, Z    +0.000, E1   +59.836, E3 +211087.431}
SPL {X  -160.000, Y  +398.875, Z    +0.000, E1   +61.100, E3 +211108.979}
SPL {X  -159.733, Y  +376.466, Z    +0.000, E1   +61.765, E3 +211130.168}
SPL {X  -158.128, Y  +361.299, Z    +0.000, E1   +61.520, E3 +211149.148}
SPL {X  -155.661, Y  +348.690, Z    +0.000, E1   +61.132, E3 +211166.104}
SPL {X  -152.251, Y  +336.510, Z    +0.000, E1   +60.617, E3 +211183.437}
SPL {X  -148.078, Y  +325.096, Z    +0.000, E1   +59.928, E3 +211200.565}
SPL {X  -143.290, Y  +314.510, Z    +0.000, E1   +59.129, E3 +211217.188}
SPL {X  -139.113, Y  +306.659, Z    +0.000, E1   +58.310, E3 +211230.039}
SPL {X  -135.700, Y  +300.932, Z    +0.000, E1   +57.683, E3 +211239.535}
SPL {X  -117.539, Y  +277.143, Z    +0.000, E1   +48.559, E3 +211354.221}
ENDSPLINE

SPLINE
SPL {X  -150.734, Y  +332.041, Z    +0.000, E1   +31.286, E3 +211456.886}
SPL {X  -159.235, Y  +370.077, Z    +0.000, E1   +12.240, E3 +211470.240}
SPL {X  -159.991, Y  +384.025, Z    +0.000, E1    +2.884, E3 +211471.789}
SPL {X  -160.000, Y  +388.170, Z    +0.000, E1    -0.470, E3 +211471.920}
SPL {X  -160.000, Y  +392.385, Z    +0.000, E1    -5.697, E3 +211472.110}
SPL {X  -160.000, Y  +398.918, Z    +0.000, E1   -15.420, E3 +211472.788}
SPL {X  -160.000, Y  +410.991, Z    +0.000, E1   -32.499, E3 +211475.284}
SPL {X  -160.000, Y  +455.466, Z    +0.000, E1   -56.407, E3 +211496.182}
SPL {X  -160.000, Y  +554.875, Z    +0.000, E1   -61.915, E3 +211578.086}
SPL {X  -160.000, Y  +571.700, Z    +0.000, E1   -61.918, E3 +211597.163}
SPL {X  -160.000, Y  +587.975, Z    +0.000, E1   -61.909, E3 +211615.630}
SPL {X  -160.000, Y  +604.690, Z    +0.000, E1   -61.922, E3 +211634.559}
SPL {X  -160.000, Y  +621.475, Z    +0.000, E1   -61.913, E3 +211653.611}
SPL {X  -160.000, Y  +638.005, Z    +0.000, E1   -61.917, E3 +211672.341}
SPL {X  -160.000, Y  +655.083, Z    +0.000, E1   -61.921, E3 +211691.703}
SPL {X  -160.000, Y  +671.910, Z    +0.000, E1   -61.915, E3 +211710.796}
SPL {X  -159.476, Y  +687.338, Z    +0.000, E1   -61.835, E3 +211728.848}
SPL {X  -157.928, Y  +700.064, Z    +0.000, E1   -61.593, E3 +211744.913}
SPL {X  -155.236, Y  +713.154, Z    +0.000, E1   -61.225, E3 +211762.460}
SPL {X  -151.860, Y  +724.785, Z    +0.000, E1   -60.654, E3 +211779.133}
SPL {X  -148.451, Y  +734.085, Z    +0.000, E1   -60.099, E3 +211793.058}
SPL {X  -144.033, Y  +744.073, Z    +0.000, E1   -59.381, E3 +211808.578}
SPL {X  -139.170, Y  +753.341, Z    +0.000, E1   -58.489, E3 +211823.600}
SPL {X  -135.320, Y  +759.772, Z    +0.000, E1   -57.727, E3 +211834.309}
SPL {X  -117.185, Y  +783.339, Z    +0.000, E1   -48.966, E3 +211942.695}
ENDSPLINE

SPLINE
SPL {X  -142.074, Y  +747.987, Z    +0.000, E1   -38.326, E3 +212041.389}
SPL {X  -154.075, Y  +717.539, Z    +0.000, E1   -26.988, E3 +212060.546}
SPL {X  -158.904, Y  +693.092, Z    +0.000, E1   -14.171, E3 +212067.337}
SPL {X  -159.937, Y  +678.885, Z    +0.000, E1    -4.971, E3 +212069.164}
SPL {X  -160.000, Y  +672.790, Z    +0.000, E1    -0.387, E3 +212069.432}
SPL {X  -160.000, Y  +669.961, Z    +0.000, E1    +2.696, E3 +212069.509}
SPL {X  -160.000, Y  +663.591, Z    +0.000, E1   +11.688, E3 +212070.003}
SPL {X  -160.000, Y  +654.521, Z    +0.000, E1   +25.997, E3 +212071.361}
SPL {X  -160.000, Y  +642.364, Z    +0.000, E1   +40.387, E3 +212074.663}
SPL {X  -160.000, Y  +597.330, Z    +0.000, E1   +58.145, E3 +212097.574}
SPL {X  -160.000, Y  +507.195, Z    +0.000, E1   +61.792, E3 +212174.905}
SPL {X  -160.000, Y  +494.139, Z    +0.000, E1   +61.770, E3 +212189.836}
SPL {X  -160.000, Y  +480.560, Z    +0.000, E1   +61.503, E3 +212207.633}
ENDSPLINE

SPLINE
SPL {X  -160.000, Y  +495.136, Z    +0.000, E1   +55.416, E3 +212229.139}
ENDSPLINE

SPLINE
SPL {X  -160.000, Y  +472.196, Z    +0.000, E1   +56.977, E3 +212251.814}
SPL {X  -160.000, Y  +448.172, Z    +0.000, E1   +58.434, E3 +212274.509}
SPL {X  -160.000, Y  +423.986, Z    +0.000, E1   +59.836, E3 +212295.762}
SPL {X  -160.000, Y  +398.875, Z    +0.000, E1   +61.100, E3 +212317.310}
SPL {X  -159.733, Y  +376.466, Z    +0.000, E1   +61.765, E3 +212338.500}
SPL {X  -158.128, Y  +361.299, Z    +0.000, E1   +61.520, E3 +212357.480}
SPL {X  -155.661, Y  +348.690, Z    +0.000, E1   +61.132, E3 +212374.436}
SPL {X  -152.251, Y  +336.510, Z    +0.000, E1   +60.617, E3 +212391.768}
SPL {X  -148.078, Y  +325.096, Z    +0.000, E1   +59.928, E3 +212408.897}
SPL {X  -143.290, Y  +314.510, Z    +0.000, E1   +59.129, E3 +212425.520}
SPL {X  -139.113, Y  +306.659, Z    +0.000, E1   +58.310, E3 +212438.371}
SPL {X  -135.700, Y  +300.932, Z    +0.000, E1   +57.683, E3 +212447.867}
SPL {X  -117.539, Y  +277.143, Z    +0.000, E1   +48.559, E3 +212562.553}
ENDSPLINE

SPLINE
SPL {X  -150.734, Y  +332.041, Z    +0.000, E1   +31.286, E3 +212665.218}
SPL {X  -159.235, Y  +370.077, Z    +0.000, E1   +12.240, E3 +212678.572}
SPL {X  -159.991, Y  +384.025, Z    +0.000, E1    +2.884, E3 +212680.121}
SPL {X  -160.000, Y  +388.170, Z    +0.000, E1    -0.470, E3 +212680.251}
SPL {X  -160.000, Y  +392.385, Z    +0.000, E1    -5.697, E3 +212680.441}
SPL {X  -160.000, Y  +398.918, Z    +0.000, E1   -15.420, E3 +212681.120}
SPL {X  -160.000, Y  +410.991, Z    +0.000, E1   -32.499, E3 +212683.615}
SPL {X  -160.000, Y  +455.466, Z    +0.000, E1   -56.407, E3 +212704.514}
SPL {X  -160.000, Y  +554.875, Z    +0.000, E1   -61.915, E3 +212786.418}
SPL {X  -160.000, Y  +571.700, Z    +0.000, E1   -61.918, E3 +212805.495}
SPL {X  -160.000, Y  +587.975, Z    +0.000, E1   -61.909, E3 +212823.961}
SPL {X  -160.000, Y  +604.690, Z    +0.000, E1   -61.922, E3 +212842.891}
SPL {X  -160.000, Y  +621.475, Z    +0.000, E1   -61.913, E3 +212861.943}
SPL {X  -160.000, Y  +638.005, Z    +0.000, E1   -61.917, E3 +212880.673}
SPL {X  -160.000, Y  +655.083, Z    +0.000, E1   -61.921, E3 +212900.034}
SPL {X  -160.000, Y  +671.910, Z    +0.000, E1   -61.915, E3 +212919.128}
SPL {X  -159.476, Y  +687.338, Z    +0.000, E1   -61.835, E3 +212937.180}
SPL {X  -157.928, Y  +700.064, Z    +0.000, E1   -61.593, E3 +212953.245}
SPL {X  -155.236, Y  +713.154, Z    +0.000, E1   -61.225, E3 +212970.792}
SPL {X  -151.860, Y  +724.785, Z    +0.000, E1   -60.654, E3 +212987.464}
SPL {X  -148.451, Y  +734.085, Z    +0.000, E1   -60.099, E3 +213001.389}
SPL {X  -144.033, Y  +744.073, Z    +0.000, E1   -59.381, E3 +213016.910}
SPL {X  -139.170, Y  +753.341, Z    +0.000, E1   -58.489, E3 +213031.931}
SPL {X  -135.320, Y  +759.772, Z    +0.000, E1   -57.727, E3 +213042.641}
SPL {X  -117.185, Y  +783.339, Z    +0.000, E1   -48.966, E3 +213151.027}
ENDSPLINE

SPLINE
SPL {X  -142.074, Y  +747.987, Z    +0.000, E1   -38.326, E3 +213249.721}
SPL {X  -154.075, Y  +717.539, Z    +0.000, E1   -26.988, E3 +213268.878}
SPL {X  -158.904, Y  +693.092, Z    +0.000, E1   -14.171, E3 +213275.669}
SPL {X  -159.937, Y  +678.885, Z    +0.000, E1    -4.971, E3 +213277.496}
SPL {X  -160.000, Y  +672.790, Z    +0.000, E1    -0.387, E3 +213277.764}
SPL {X  -160.000, Y  +669.961, Z    +0.000, E1    +2.696, E3 +213277.841}
SPL {X  -160.000, Y  +663.591, Z    +0.000, E1   +11.688, E3 +213278.335}
SPL {X  -160.000, Y  +654.521, Z    +0.000, E1   +25.997, E3 +213279.693}
SPL {X  -160.000, Y  +642.364, Z    +0.000, E1   +40.387, E3 +213282.995}
SPL {X  -160.000, Y  +597.330, Z    +0.000, E1   +58.145, E3 +213305.906}
SPL {X  -160.000, Y  +507.195, Z    +0.000, E1   +61.792, E3 +213383.237}
SPL {X  -160.000, Y  +494.139, Z    +0.000, E1   +61.770, E3 +213398.167}
SPL {X  -160.000, Y  +480.560, Z    +0.000, E1   +61.503, E3 +213415.964}
ENDSPLINE

SPLINE
SPL {X  -160.000, Y  +495.136, Z    +0.000, E1   +55.416, E3 +213437.471}
ENDSPLINE

SPLINE
SPL {X  -160.000, Y  +472.196, Z    +0.000, E1   +56.977, E3 +213460.146}
SPL {X  -160.000, Y  +448.172, Z    +0.000, E1   +58.434, E3 +213482.841}
SPL {X  -160.000, Y  +423.986, Z    +0.000, E1   +59.836, E3 +213504.094}
SPL {X  -160.000, Y  +398.875, Z    +0.000, E1   +61.100, E3 +213525.642}
SPL {X  -159.733, Y  +376.466, Z    +0.000, E1   +61.765, E3 +213546.832}
SPL {X  -158.128, Y  +361.299, Z    +0.000, E1   +61.520, E3 +213565.811}
SPL {X  -155.661, Y  +348.690, Z    +0.000, E1   +61.132, E3 +213582.767}
SPL {X  -152.251, Y  +336.510, Z    +0.000, E1   +60.617, E3 +213600.100}
SPL {X  -148.078, Y  +325.096, Z    +0.000, E1   +59.928, E3 +213617.229}
SPL {X  -143.290, Y  +314.510, Z    +0.000, E1   +59.129, E3 +213633.852}
SPL {X  -139.113, Y  +306.659, Z    +0.000, E1   +58.310, E3 +213646.702}
SPL {X  -135.700, Y  +300.932, Z    +0.000, E1   +57.683, E3 +213656.199}
SPL {X  -117.539, Y  +277.143, Z    +0.000, E1   +48.559, E3 +213770.885}
ENDSPLINE

SPLINE
SPL {X  -150.734, Y  +332.041, Z    +0.000, E1   +31.286, E3 +213873.550}
SPL {X  -159.235, Y  +370.077, Z    +0.000, E1   +12.240, E3 +213886.904}
SPL {X  -159.991, Y  +384.025, Z    +0.000, E1    +2.884, E3 +213888.452}
SPL {X  -160.000, Y  +388.170, Z    +0.000, E1    -0.470, E3 +213888.583}
SPL {X  -160.000, Y  +392.385, Z    +0.000, E1    -5.697, E3 +213888.773}
SPL {X  -160.000, Y  +398.918, Z    +0.000, E1   -15.420, E3 +213889.452}
SPL {X  -160.000, Y  +410.991, Z    +0.000, E1   -32.499, E3 +213891.947}
SPL {X  -160.000, Y  +455.466, Z    +0.000, E1   -56.407, E3 +213912.846}
SPL {X  -160.000, Y  +554.875, Z    +0.000, E1   -61.915, E3 +213994.750}
SPL {X  -160.000, Y  +571.700, Z    +0.000, E1   -61.918, E3 +214013.827}
SPL {X  -160.000, Y  +587.975, Z    +0.000, E1   -61.909, E3 +214032.293}
SPL {X  -160.000, Y  +604.690, Z    +0.000, E1   -61.922, E3 +214051.222}
SPL {X  -160.000, Y  +621.475, Z    +0.000, E1   -61.913, E3 +214070.274}
SPL {X  -160.000, Y  +638.005, Z    +0.000, E1   -61.917, E3 +214089.005}
SPL {X  -160.000, Y  +655.083, Z    +0.000, E1   -61.921, E3 +214108.366}
SPL {X  -160.000, Y  +671.910, Z    +0.000, E1   -61.915, E3 +214127.460}
SPL {X  -159.476, Y  +687.338, Z    +0.000, E1   -61.835, E3 +214145.512}
SPL {X  -157.928, Y  +700.064, Z    +0.000, E1   -61.593, E3 +214161.576}
SPL {X  -155.236, Y  +713.154, Z    +0.000, E1   -61.225, E3 +214179.124}
SPL {X  -151.860, Y  +724.785, Z    +0.000, E1   -60.654, E3 +214195.796}
SPL {X  -148.451, Y  +734.085, Z    +0.000, E1   -60.099, E3 +214209.721}
SPL {X  -144.033, Y  +744.073, Z    +0.000, E1   -59.381, E3 +214225.242}
SPL {X  -139.170, Y  +753.341, Z    +0.000, E1   -58.489, E3 +214240.263}
SPL {X  -135.320, Y  +759.772, Z    +0.000, E1   -57.727, E3 +214250.973}
SPL {X  -117.185, Y  +783.339, Z    +0.000, E1   -48.966, E3 +214359.359}
ENDSPLINE

SPLINE
SPL {X  -142.074, Y  +747.987, Z    +0.000, E1   -38.326, E3 +214458.052}
SPL {X  -154.075, Y  +717.539, Z    +0.000, E1   -26.988, E3 +214477.209}
SPL {X  -158.904, Y  +693.092, Z    +0.000, E1   -14.171, E3 +214484.001}
SPL {X  -159.937, Y  +678.885, Z    +0.000, E1    -4.971, E3 +214485.828}
SPL {X  -160.000, Y  +672.790, Z    +0.000, E1    -0.387, E3 +214486.096}
SPL {X  -160.000, Y  +669.961, Z    +0.000, E1    +2.696, E3 +214486.172}
SPL {X  -160.000, Y  +663.591, Z    +0.000, E1   +11.688, E3 +214486.667}
SPL {X  -160.000, Y  +654.521, Z    +0.000, E1   +25.997, E3 +214488.025}
SPL {X  -160.000, Y  +642.364, Z    +0.000, E1   +40.387, E3 +214491.327}
SPL {X  -160.000, Y  +597.330, Z    +0.000, E1   +58.145, E3 +214514.238}
SPL {X  -160.000, Y  +507.195, Z    +0.000, E1   +61.792, E3 +214591.569}
SPL {X  -160.000, Y  +494.139, Z    +0.000, E1   +61.770, E3 +214606.499}
SPL {X  -160.000, Y  +480.560, Z    +0.000, E1   +61.503, E3 +214624.296}
ENDSPLINE

SPLINE
SPL {X  -160.000, Y  +495.136, Z    +0.000, E1   +55.416, E3 +214645.803}
ENDSPLINE

SPLINE
SPL {X  -160.000, Y  +472.196, Z    +0.000, E1   +56.977, E3 +214668.478}
SPL {X  -160.000, Y  +448.172, Z    +0.000, E1   +58.434, E3 +214691.172}
SPL {X  -160.000, Y  +423.986, Z    +0.000, E1   +59.836, E3 +214712.426}
SPL {X  -160.000, Y  +398.875, Z    +0.000, E1   +61.100, E3 +214733.974}
SPL {X  -159.733, Y  +376.466, Z    +0.000, E1   +61.765, E3 +214755.164}
SPL {X  -158.128, Y  +361.299, Z    +0.000, E1   +61.520, E3 +214774.143}
SPL {X  -155.661, Y  +348.690, Z    +0.000, E1   +61.132, E3 +214791.099}
SPL {X  -152.251, Y  +336.510, Z    +0.000, E1   +60.617, E3 +214808.432}
SPL {X  -148.078, Y  +325.096, Z    +0.000, E1   +59.928, E3 +214825.560}
SPL {X  -143.290, Y  +314.510, Z    +0.000, E1   +59.129, E3 +214842.183}
SPL {X  -139.113, Y  +306.659, Z    +0.000, E1   +58.310, E3 +214855.034}
SPL {X  -135.700, Y  +300.932, Z    +0.000, E1   +57.683, E3 +214864.531}
SPL {X  -117.539, Y  +277.143, Z    +0.000, E1   +48.559, E3 +214979.217}
ENDSPLINE

SPLINE
SPL {X  -150.734, Y  +332.041, Z    +0.000, E1   +31.286, E3 +215081.881}
SPL {X  -159.235, Y  +370.077, Z    +0.000, E1   +12.240, E3 +215095.236}
SPL {X  -159.991, Y  +384.025, Z    +0.000, E1    +2.884, E3 +215096.784}
SPL {X  -160.000, Y  +388.170, Z    +0.000, E1    -0.470, E3 +215096.915}
SPL {X  -160.000, Y  +392.385, Z    +0.000, E1    -5.697, E3 +215097.105}
SPL {X  -160.000, Y  +398.918, Z    +0.000, E1   -15.420, E3 +215097.784}
SPL {X  -160.000, Y  +410.991, Z    +0.000, E1   -32.499, E3 +215100.279}
SPL {X  -160.000, Y  +455.466, Z    +0.000, E1   -56.407, E3 +215121.178}
SPL {X  -160.000, Y  +554.875, Z    +0.000, E1   -61.915, E3 +215203.081}
SPL {X  -160.000, Y  +571.700, Z    +0.000, E1   -61.918, E3 +215222.158}
SPL {X  -160.000, Y  +587.975, Z    +0.000, E1   -61.909, E3 +215240.625}
SPL {X  -160.000, Y  +604.690, Z    +0.000, E1   -61.922, E3 +215259.554}
SPL {X  -160.000, Y  +621.475, Z    +0.000, E1   -61.913, E3 +215278.606}
SPL {X  -160.000, Y  +638.005, Z    +0.000, E1   -61.917, E3 +215297.336}
SPL {X  -160.000, Y  +655.083, Z    +0.000, E1   -61.921, E3 +215316.698}
SPL {X  -160.000, Y  +671.910, Z    +0.000, E1   -61.915, E3 +215335.792}
SPL {X  -159.476, Y  +687.338, Z    +0.000, E1   -61.835, E3 +215353.844}
SPL {X  -157.928, Y  +700.064, Z    +0.000, E1   -61.593, E3 +215369.908}
SPL {X  -155.236, Y  +713.154, Z    +0.000, E1   -61.225, E3 +215387.455}
SPL {X  -151.860, Y  +724.785, Z    +0.000, E1   -60.654, E3 +215404.128}
SPL {X  -148.451, Y  +734.085, Z    +0.000, E1   -60.099, E3 +215418.053}
SPL {X  -144.033, Y  +744.073, Z    +0.000, E1   -59.381, E3 +215433.573}
SPL {X  -139.170, Y  +753.341, Z    +0.000, E1   -58.489, E3 +215448.595}
SPL {X  -135.320, Y  +759.772, Z    +0.000, E1   -57.727, E3 +215459.304}
SPL {X  -117.185, Y  +783.339, Z    +0.000, E1   -48.966, E3 +215567.691}
ENDSPLINE

SPLINE
SPL {X  -142.074, Y  +747.987, Z    +0.000, E1   -38.326, E3 +215666.384}
SPL {X  -154.075, Y  +717.539, Z    +0.000, E1   -26.988, E3 +215685.541}
SPL {X  -158.904, Y  +693.092, Z    +0.000, E1   -14.171, E3 +215692.332}
SPL {X  -159.937, Y  +678.885, Z    +0.000, E1    -4.971, E3 +215694.160}
SPL {X  -160.000, Y  +672.790, Z    +0.000, E1    -0.387, E3 +215694.427}
SPL {X  -160.000, Y  +669.961, Z    +0.000, E1    +2.696, E3 +215694.504}
SPL {X  -160.000, Y  +663.591, Z    +0.000, E1   +11.688, E3 +215694.998}
SPL {X  -160.000, Y  +654.521, Z    +0.000, E1   +25.997, E3 +215696.356}
SPL {X  -160.000, Y  +642.364, Z    +0.000, E1   +40.387, E3 +215699.658}
SPL {X  -160.000, Y  +597.330, Z    +0.000, E1   +58.145, E3 +215722.570}
SPL {X  -160.000, Y  +516.293, Z    +0.000, E1   +61.751, E3 +215789.627}
SPL {X  -160.000, Y  +506.292, Z    +0.000, E1   +61.780, E3 +215800.961}
SPL {X  -160.000, Y  +494.139, Z    +0.000, E1   +61.770, E3 +215814.831}
SPL {X  -160.000, Y  +480.560, Z    +0.000, E1   +61.503, E3 +215832.628}
ENDSPLINE

SPLINE
SPL {X  -160.000, Y  +495.136, Z    +0.000, E1   +55.416, E3 +215854.135}
ENDSPLINE

SPLINE
SPL {X  -160.000, Y  +472.196, Z    +0.000, E1   +56.977, E3 +215876.809}
SPL {X  -160.000, Y  +448.172, Z    +0.000, E1   +58.434, E3 +215899.504}
SPL {X  -160.000, Y  +423.986, Z    +0.000, E1   +59.836, E3 +215920.758}
SPL {X  -160.000, Y  +398.875, Z    +0.000, E1   +61.100, E3 +215942.306}
SPL {X  -159.733, Y  +376.466, Z    +0.000, E1   +61.765, E3 +215963.495}
SPL {X  -158.128, Y  +361.299, Z    +0.000, E1   +61.520, E3 +215982.475}
SPL {X  -155.661, Y  +348.690, Z    +0.000, E1   +61.132, E3 +215999.431}
SPL {X  -152.251, Y  +336.510, Z    +0.000, E1   +60.617, E3 +216016.764}
SPL {X  -148.078, Y  +325.096, Z    +0.000, E1   +59.928, E3 +216033.892}
SPL {X  -143.290, Y  +314.510, Z    +0.000, E1   +59.129, E3 +216050.515}
SPL {X  -139.113, Y  +306.659, Z    +0.000, E1   +58.310, E3 +216063.366}
SPL {X  -135.700, Y  +300.932, Z    +0.000, E1   +57.683, E3 +216072.862}
SPL {X  -117.539, Y  +277.143, Z    +0.000, E1   +48.559, E3 +216187.548}
ENDSPLINE

SPLINE
SPL {X  -150.734, Y  +332.041, Z    +0.000, E1   +31.286, E3 +216290.213}
SPL {X  -159.235, Y  +370.077, Z    +0.000, E1   +12.240, E3 +216303.567}
SPL {X  -159.991, Y  +384.025, Z    +0.000, E1    +2.884, E3 +216305.116}
SPL {X  -160.000, Y  +388.170, Z    +0.000, E1    -0.470, E3 +216305.247}
SPL {X  -160.000, Y  +392.385, Z    +0.000, E1    -5.697, E3 +216305.437}
SPL {X  -160.000, Y  +398.918, Z    +0.000, E1   -15.420, E3 +216306.115}
SPL {X  -160.000, Y  +410.991, Z    +0.000, E1   -32.499, E3 +216308.611}
SPL {X  -160.000, Y  +455.466, Z    +0.000, E1   -56.407, E3 +216329.509}
SPL {X  -160.000, Y  +554.875, Z    +0.000, E1   -61.915, E3 +216411.413}
SPL {X  -160.000, Y  +571.700, Z    +0.000, E1   -61.918, E3 +216430.490}
SPL {X  -160.000, Y  +587.975, Z    +0.000, E1   -61.909, E3 +216448.957}
SPL {X  -160.000, Y  +604.690, Z    +0.000, E1   -61.922, E3 +216467.886}
SPL {X  -160.000, Y  +621.475, Z    +0.000, E1   -61.913, E3 +216486.938}
SPL {X  -160.000, Y  +638.005, Z    +0.000, E1   -61.917, E3 +216505.668}
SPL {X  -160.000, Y  +655.083, Z    +0.000, E1   -61.921, E3 +216525.030}
SPL {X  -160.000, Y  +671.910, Z    +0.000, E1   -61.915, E3 +216544.123}
SPL {X  -159.476, Y  +687.338, Z    +0.000, E1   -61.835, E3 +216562.175}
SPL {X  -157.928, Y  +700.064, Z    +0.000, E1   -61.593, E3 +216578.240}
SPL {X  -155.236, Y  +713.154, Z    +0.000, E1   -61.225, E3 +216595.787}
SPL {X  -151.860, Y  +724.785, Z    +0.000, E1   -60.654, E3 +216612.460}
SPL {X  -148.451, Y  +734.085, Z    +0.000, E1   -60.099, E3 +216626.385}
SPL {X  -144.033, Y  +744.073, Z    +0.000, E1   -59.381, E3 +216641.905}
SPL {X  -139.170, Y  +753.341, Z    +0.000, E1   -58.489, E3 +216656.927}
SPL {X  -135.320, Y  +759.772, Z    +0.000, E1   -57.727, E3 +216667.636}
SPL {X  -117.185, Y  +783.339, Z    +0.000, E1   -48.966, E3 +216776.022}
ENDSPLINE

SPLINE
SPL {X  -142.074, Y  +747.987, Z    +0.000, E1   -38.326, E3 +216874.716}
SPL {X  -154.075, Y  +717.539, Z    +0.000, E1   -26.988, E3 +216893.873}
SPL {X  -158.904, Y  +693.092, Z    +0.000, E1   -14.171, E3 +216900.664}
SPL {X  -159.937, Y  +678.885, Z    +0.000, E1    -4.971, E3 +216902.491}
SPL {X  -160.000, Y  +672.790, Z    +0.000, E1    -0.387, E3 +216902.759}
SPL {X  -160.000, Y  +669.961, Z    +0.000, E1    +2.696, E3 +216902.836}
SPL {X  -160.000, Y  +663.591, Z    +0.000, E1   +11.688, E3 +216903.330}
SPL {X  -160.000, Y  +654.521, Z    +0.000, E1   +25.997, E3 +216904.688}
SPL {X  -160.000, Y  +642.364, Z    +0.000, E1   +40.387, E3 +216907.990}
SPL {X  -160.000, Y  +597.330, Z    +0.000, E1   +58.145, E3 +216930.901}
SPL {X  -160.000, Y  +507.195, Z    +0.000, E1   +61.792, E3 +217008.232}
SPL {X  -160.000, Y  +494.139, Z    +0.000, E1   +61.770, E3 +217023.163}
SPL {X  -160.000, Y  +480.560, Z    +0.000, E1   +61.503, E3 +217040.960}
ENDSPLINE

SPLINE
SPL {X  -160.000, Y  +495.136, Z    +0.000, E1   +55.416, E3 +217062.466}
ENDSPLINE

SPLINE
SPL {X  -160.000, Y  +472.196, Z    +0.000, E1   +56.977, E3 +217085.141}
SPL {X  -160.000, Y  +448.172, Z    +0.000, E1   +58.434, E3 +217107.836}
SPL {X  -160.000, Y  +423.986, Z    +0.000, E1   +59.836, E3 +217129.090}
SPL {X  -160.000, Y  +398.875, Z    +0.000, E1   +61.100, E3 +217150.638}
SPL {X  -159.733, Y  +376.466, Z    +0.000, E1   +61.765, E3 +217171.827}
SPL {X  -158.128, Y  +361.299, Z    +0.000, E1   +61.520, E3 +217190.807}
SPL {X  -155.661, Y  +348.690, Z    +0.000, E1   +61.132, E3 +217207.763}
SPL {X  -152.251, Y  +336.510, Z    +0.000, E1   +60.617, E3 +217225.096}
SPL {X  -148.078, Y  +325.096, Z    +0.000, E1   +59.928, E3 +217242.224}
SPL {X  -143.290, Y  +314.510, Z    +0.000, E1   +59.129, E3 +217258.847}
SPL {X  -139.113, Y  +306.659, Z    +0.000, E1   +58.310, E3 +217271.698}
SPL {X  -135.700, Y  +300.932, Z    +0.000, E1   +57.683, E3 +217281.194}
SPL {X  -117.539, Y  +277.143, Z    +0.000, E1   +48.559, E3 +217395.880}
ENDSPLINE

SPLINE
SPL {X  -150.734, Y  +332.041, Z    +0.000, E1   +31.286, E3 +217498.545}
SPL {X  -159.235, Y  +370.077, Z    +0.000, E1   +12.240, E3 +217511.899}
SPL {X  -159.991, Y  +384.025, Z    +0.000, E1    +2.884, E3 +217513.448}
SPL {X  -160.000, Y  +388.170, Z    +0.000, E1    -0.470, E3 +217513.578}
SPL {X  -160.000, Y  +392.385, Z    +0.000, E1    -5.697, E3 +217513.769}
SPL {X  -160.000, Y  +398.918, Z    +0.000, E1   -15.420, E3 +217514.447}
SPL {X  -160.000, Y  +410.991, Z    +0.000, E1   -32.499, E3 +217516.942}
SPL {X  -160.000, Y  +455.466, Z    +0.000, E1   -56.407, E3 +217537.841}
SPL {X  -160.000, Y  +554.875, Z    +0.000, E1   -61.915, E3 +217619.745}
SPL {X  -160.000, Y  +571.700, Z    +0.000, E1   -61.918, E3 +217638.822}
SPL {X  -160.000, Y  +587.975, Z    +0.000, E1   -61.909, E3 +217657.288}
SPL {X  -160.000, Y  +604.690, Z    +0.000, E1   -61.922, E3 +217676.218}
SPL {X  -160.000, Y  +621.475, Z    +0.000, E1   -61.913, E3 +217695.270}
SPL {X  -160.000, Y  +638.005, Z    +0.000, E1   -61.917, E3 +217714.000}
SPL {X  -160.000, Y  +655.083, Z    +0.000, E1   -61.921, E3 +217733.361}
SPL {X  -160.000, Y  +671.910, Z    +0.000, E1   -61.915, E3 +217752.455}
SPL {X  -159.476, Y  +687.338, Z    +0.000, E1   -61.835, E3 +217770.507}
SPL {X  -157.928, Y  +700.064, Z    +0.000, E1   -61.593, E3 +217786.572}
SPL {X  -155.236, Y  +713.154, Z    +0.000, E1   -61.225, E3 +217804.119}
SPL {X  -151.860, Y  +724.785, Z    +0.000, E1   -60.654, E3 +217820.791}
SPL {X  -148.451, Y  +734.085, Z    +0.000, E1   -60.099, E3 +217834.716}
SPL {X  -144.033, Y  +744.073, Z    +0.000, E1   -59.381, E3 +217850.237}
SPL {X  -139.170, Y  +753.341, Z    +0.000, E1   -58.489, E3 +217865.258}
SPL {X  -135.320, Y  +759.772, Z    +0.000, E1   -57.727, E3 +217875.968}
SPL {X  -117.185, Y  +783.339, Z    +0.000, E1   -48.966, E3 +217984.354}
ENDSPLINE

SPLINE
SPL {X  -142.074, Y  +747.987, Z    +0.000, E1   -38.326, E3 +218083.048}
SPL {X  -154.075, Y  +717.539, Z    +0.000, E1   -26.988, E3 +218102.205}
SPL {X  -158.904, Y  +693.092, Z    +0.000, E1   -14.171, E3 +218108.996}
SPL {X  -159.937, Y  +678.885, Z    +0.000, E1    -4.971, E3 +218110.823}
SPL {X  -160.000, Y  +672.790, Z    +0.000, E1    -0.387, E3 +218111.091}
SPL {X  -160.000, Y  +669.961, Z    +0.000, E1    +2.696, E3 +218111.168}
SPL {X  -160.000, Y  +663.591, Z    +0.000, E1   +11.688, E3 +218111.662}
SPL {X  -160.000, Y  +654.521, Z    +0.000, E1   +25.997, E3 +218113.020}
SPL {X  -160.000, Y  +642.364, Z    +0.000, E1   +40.387, E3 +218116.322}
SPL {X  -160.000, Y  +597.330, Z    +0.000, E1   +58.145, E3 +218139.233}
SPL {X  -160.000, Y  +507.195, Z    +0.000, E1   +61.792, E3 +218216.564}
SPL {X  -160.000, Y  +494.139, Z    +0.000, E1   +61.770, E3 +218231.494}
SPL {X  -160.000, Y  +480.560, Z    +0.000, E1   +61.503, E3 +218249.291}
ENDSPLINE

SPLINE
SPL {X  -160.000, Y  +495.136, Z    +0.000, E1   +55.416, E3 +218270.798}
ENDSPLINE

SPLINE
SPL {X  -160.000, Y  +472.196, Z    +0.000, E1   +56.977, E3 +218293.473}
SPL {X  -160.000, Y  +448.172, Z    +0.000, E1   +58.434, E3 +218316.168}
SPL {X  -160.000, Y  +423.986, Z    +0.000, E1   +59.836, E3 +218337.421}
SPL {X  -160.000, Y  +398.875, Z    +0.000, E1   +61.100, E3 +218358.969}
SPL {X  -159.733, Y  +376.466, Z    +0.000, E1   +61.765, E3 +218380.159}
SPL {X  -158.128, Y  +361.299, Z    +0.000, E1   +61.520, E3 +218399.138}
SPL {X  -155.661, Y  +348.690, Z    +0.000, E1   +61.132, E3 +218416.095}
SPL {X  -152.251, Y  +336.510, Z    +0.000, E1   +60.617, E3 +218433.427}
SPL {X  -148.078, Y  +325.096, Z    +0.000, E1   +59.928, E3 +218450.556}
SPL {X  -143.290, Y  +314.510, Z    +0.000, E1   +59.129, E3 +218467.179}
SPL {X  -139.113, Y  +306.659, Z    +0.000, E1   +58.310, E3 +218480.029}
SPL {X  -135.700, Y  +300.932, Z    +0.000, E1   +57.683, E3 +218489.526}
SPL {X  -117.539, Y  +277.143, Z    +0.000, E1   +48.559, E3 +218604.212}
ENDSPLINE

SPLINE
SPL {X  -150.734, Y  +332.041, Z    +0.000, E1   +31.286, E3 +218706.877}
SPL {X  -159.235, Y  +370.077, Z    +0.000, E1   +12.240, E3 +218720.231}
SPL {X  -159.991, Y  +384.025, Z    +0.000, E1    +2.884, E3 +218721.780}
SPL {X  -160.000, Y  +388.170, Z    +0.000, E1    -0.470, E3 +218721.910}
SPL {X  -160.000, Y  +392.385, Z    +0.000, E1    -5.697, E3 +218722.100}
SPL {X  -160.000, Y  +398.918, Z    +0.000, E1   -15.420, E3 +218722.779}
SPL {X  -160.000, Y  +410.991, Z    +0.000, E1   -32.499, E3 +218725.274}
SPL {X  -160.000, Y  +455.466, Z    +0.000, E1   -56.407, E3 +218746.173}
SPL {X  -160.000, Y  +554.875, Z    +0.000, E1   -61.915, E3 +218828.077}
SPL {X  -160.000, Y  +571.700, Z    +0.000, E1   -61.918, E3 +218847.154}
SPL {X  -160.000, Y  +587.975, Z    +0.000, E1   -61.909, E3 +218865.620}
SPL {X  -160.000, Y  +604.690, Z    +0.000, E1   -61.922, E3 +218884.549}
SPL {X  -160.000, Y  +621.475, Z    +0.000, E1   -61.913, E3 +218903.601}
SPL {X  -160.000, Y  +638.005, Z    +0.000, E1   -61.917, E3 +218922.332}
SPL {X  -160.000, Y  +655.083, Z    +0.000, E1   -61.921, E3 +218941.693}
SPL {X  -160.000, Y  +671.910, Z    +0.000, E1   -61.915, E3 +218960.787}
SPL {X  -159.476, Y  +687.338, Z    +0.000, E1   -61.835, E3 +218978.839}
SPL {X  -157.928, Y  +700.064, Z    +0.000, E1   -61.593, E3 +218994.903}
SPL {X  -155.236, Y  +713.154, Z    +0.000, E1   -61.225, E3 +219012.451}
SPL {X  -151.860, Y  +724.785, Z    +0.000, E1   -60.654, E3 +219029.123}
SPL {X  -148.451, Y  +734.085, Z    +0.000, E1   -60.099, E3 +219043.048}
SPL {X  -144.033, Y  +744.073, Z    +0.000, E1   -59.381, E3 +219058.569}
SPL {X  -139.170, Y  +753.341, Z    +0.000, E1   -58.489, E3 +219073.590}
SPL {X  -135.320, Y  +759.772, Z    +0.000, E1   -57.727, E3 +219084.300}
SPL {X  -117.185, Y  +783.339, Z    +0.000, E1   -48.966, E3 +219192.686}
ENDSPLINE

SPLINE
SPL {X  -142.074, Y  +747.987, Z    +0.000, E1   -38.326, E3 +219291.379}
SPL {X  -154.075, Y  +717.539, Z    +0.000, E1   -26.988, E3 +219310.537}
SPL {X  -158.904, Y  +693.092, Z    +0.000, E1   -14.171, E3 +219317.328}
SPL {X  -159.937, Y  +678.885, Z    +0.000, E1    -4.971, E3 +219319.155}
SPL {X  -160.000, Y  +672.790, Z    +0.000, E1    -0.387, E3 +219319.423}
SPL {X  -160.000, Y  +669.961, Z    +0.000, E1    +2.696, E3 +219319.499}
SPL {X  -160.000, Y  +663.591, Z    +0.000, E1   +11.688, E3 +219319.994}
SPL {X  -160.000, Y  +654.521, Z    +0.000, E1   +25.997, E3 +219321.352}
SPL {X  -160.000, Y  +642.364, Z    +0.000, E1   +40.387, E3 +219324.654}
SPL {X  -160.000, Y  +597.330, Z    +0.000, E1   +58.145, E3 +219347.565}
SPL {X  -160.000, Y  +507.195, Z    +0.000, E1   +61.792, E3 +219424.896}
SPL {X  -160.000, Y  +494.139, Z    +0.000, E1   +61.770, E3 +219439.826}
SPL {X  -160.000, Y  +480.560, Z    +0.000, E1   +61.503, E3 +219457.623}
ENDSPLINE

SPLINE
SPL {X  -160.000, Y  +495.136, Z    +0.000, E1   +55.416, E3 +219479.130}
ENDSPLINE

SPLINE
SPL {X  -160.000, Y  +472.196, Z    +0.000, E1   +56.977, E3 +219501.805}
SPL {X  -160.000, Y  +448.172, Z    +0.000, E1   +58.434, E3 +219524.499}
SPL {X  -160.000, Y  +423.986, Z    +0.000, E1   +59.836, E3 +219545.753}
SPL {X  -160.000, Y  +398.875, Z    +0.000, E1   +61.100, E3 +219567.301}
SPL {X  -159.733, Y  +376.466, Z    +0.000, E1   +61.765, E3 +219588.491}
SPL {X  -158.128, Y  +361.299, Z    +0.000, E1   +61.520, E3 +219607.470}
SPL {X  -155.661, Y  +348.690, Z    +0.000, E1   +61.132, E3 +219624.426}
SPL {X  -152.251, Y  +336.510, Z    +0.000, E1   +60.617, E3 +219641.759}
SPL {X  -148.078, Y  +325.096, Z    +0.000, E1   +59.928, E3 +219658.888}
SPL {X  -143.290, Y  +314.510, Z    +0.000, E1   +59.129, E3 +219675.510}
SPL {X  -139.113, Y  +306.659, Z    +0.000, E1   +58.310, E3 +219688.361}
SPL {X  -135.700, Y  +300.932, Z    +0.000, E1   +57.683, E3 +219697.858}
SPL {X  -117.539, Y  +277.143, Z    +0.000, E1   +48.559, E3 +219812.544}
ENDSPLINE

SPLINE
SPL {X  -150.734, Y  +332.041, Z    +0.000, E1   +31.286, E3 +219915.208}
SPL {X  -159.235, Y  +370.077, Z    +0.000, E1   +12.240, E3 +219928.563}
SPL {X  -159.991, Y  +384.025, Z    +0.000, E1    +2.884, E3 +219930.111}
SPL {X  -160.000, Y  +388.170, Z    +0.000, E1    -0.470, E3 +219930.242}
SPL {X  -160.000, Y  +392.385, Z    +0.000, E1    -5.697, E3 +219930.432}
SPL {X  -160.000, Y  +398.918, Z    +0.000, E1   -15.420, E3 +219931.111}
SPL {X  -160.000, Y  +410.991, Z    +0.000, E1   -32.499, E3 +219933.606}
SPL {X  -160.000, Y  +455.466, Z    +0.000, E1   -56.407, E3 +219954.505}
SPL {X  -160.000, Y  +554.875, Z    +0.000, E1   -61.915, E3 +220036.409}
SPL {X  -160.000, Y  +571.700, Z    +0.000, E1   -61.918, E3 +220055.485}
SPL {X  -160.000, Y  +587.975, Z    +0.000, E1   -61.909, E3 +220073.952}
SPL {X  -160.000, Y  +604.690, Z    +0.000, E1   -61.922, E3 +220092.881}
SPL {X  -160.000, Y  +621.475, Z    +0.000, E1   -61.913, E3 +220111.933}
SPL {X  -160.000, Y  +638.005, Z    +0.000, E1   -61.917, E3 +220130.663}
SPL {X  -160.000, Y  +655.083, Z    +0.000, E1   -61.921, E3 +220150.025}
SPL {X  -160.000, Y  +671.910, Z    +0.000, E1   -61.915, E3 +220169.119}
SPL {X  -159.476, Y  +687.338, Z    +0.000, E1   -61.835, E3 +220187.171}
SPL {X  -157.928, Y  +700.064, Z    +0.000, E1   -61.593, E3 +220203.235}
SPL {X  -155.236, Y  +713.154, Z    +0.000, E1   -61.225, E3 +220220.782}
SPL {X  -151.860, Y  +724.785, Z    +0.000, E1   -60.654, E3 +220237.455}
SPL {X  -148.451, Y  +734.085, Z    +0.000, E1   -60.099, E3 +220251.380}
SPL {X  -144.033, Y  +744.073, Z    +0.000, E1   -59.381, E3 +220266.900}
SPL {X  -139.170, Y  +753.341, Z    +0.000, E1   -58.489, E3 +220281.922}
SPL {X  -135.320, Y  +759.772, Z    +0.000, E1   -57.727, E3 +220292.631}
SPL {X  -117.185, Y  +783.339, Z    +0.000, E1   -48.966, E3 +220401.018}
ENDSPLINE

SPLINE
SPL {X  -142.074, Y  +747.987, Z    +0.000, E1   -38.326, E3 +220499.711}
SPL {X  -154.075, Y  +717.539, Z    +0.000, E1   -26.988, E3 +220518.868}
SPL {X  -158.904, Y  +693.092, Z    +0.000, E1   -14.171, E3 +220525.659}
SPL {X  -159.937, Y  +678.885, Z    +0.000, E1    -4.971, E3 +220527.487}
SPL {X  -160.000, Y  +672.790, Z    +0.000, E1    -0.387, E3 +220527.754}
SPL {X  -160.000, Y  +669.961, Z    +0.000, E1    +2.696, E3 +220527.831}
SPL {X  -160.000, Y  +663.591, Z    +0.000, E1   +11.688, E3 +220528.325}
SPL {X  -160.000, Y  +654.521, Z    +0.000, E1   +25.997, E3 +220529.683}
SPL {X  -160.000, Y  +642.364, Z    +0.000, E1   +40.387, E3 +220532.985}
SPL {X  -160.000, Y  +597.330, Z    +0.000, E1   +58.145, E3 +220555.897}
SPL {X  -160.000, Y  +516.293, Z    +0.000, E1   +61.751, E3 +220622.954}
SPL {X  -160.000, Y  +506.292, Z    +0.000, E1   +61.780, E3 +220634.288}
SPL {X  -160.000, Y  +494.139, Z    +0.000, E1   +61.770, E3 +220648.158}
SPL {X  -160.000, Y  +480.560, Z    +0.000, E1   +61.503, E3 +220665.955}
ENDSPLINE

SPLINE
SPL {X  -160.000, Y  +495.136, Z    +0.000, E1   +55.416, E3 +220687.462}
ENDSPLINE

SPLINE
SPL {X  -160.000, Y  +472.196, Z    +0.000, E1   +56.977, E3 +220710.136}
SPL {X  -160.000, Y  +448.172, Z    +0.000, E1   +58.434, E3 +220732.831}
SPL {X  -160.000, Y  +423.986, Z    +0.000, E1   +59.836, E3 +220754.085}
SPL {X  -160.000, Y  +398.875, Z    +0.000, E1   +61.100, E3 +220775.633}
SPL {X  -159.733, Y  +376.466, Z    +0.000, E1   +61.765, E3 +220796.822}
SPL {X  -158.128, Y  +361.299, Z    +0.000, E1   +61.520, E3 +220815.802}
SPL {X  -155.661, Y  +348.690, Z    +0.000, E1   +61.132, E3 +220832.758}
SPL {X  -152.251, Y  +336.510, Z    +0.000, E1   +60.617, E3 +220850.091}
SPL {X  -148.078, Y  +325.096, Z    +0.000, E1   +59.928, E3 +220867.219}
SPL {X  -143.290, Y  +314.510, Z    +0.000, E1   +59.129, E3 +220883.842}
SPL {X  -139.113, Y  +306.659, Z    +0.000, E1   +58.310, E3 +220896.693}
SPL {X  -135.700, Y  +300.932, Z    +0.000, E1   +57.683, E3 +220906.189}
SPL {X  -117.539, Y  +277.143, Z    +0.000, E1   +48.559, E3 +221020.875}
ENDSPLINE

SPLINE
SPL {X  -150.734, Y  +332.041, Z    +0.000, E1   +31.286, E3 +221123.540}
SPL {X  -159.235, Y  +370.077, Z    +0.000, E1   +12.240, E3 +221136.894}
SPL {X  -159.991, Y  +384.025, Z    +0.000, E1    +2.884, E3 +221138.443}
SPL {X  -160.000, Y  +388.170, Z    +0.000, E1    -0.470, E3 +221138.574}
SPL {X  -160.000, Y  +392.385, Z    +0.000, E1    -5.697, E3 +221138.764}
SPL {X  -160.000, Y  +398.918, Z    +0.000, E1   -15.420, E3 +221139.442}
SPL {X  -160.000, Y  +410.991, Z    +0.000, E1   -32.499, E3 +221141.938}
SPL {X  -160.000, Y  +455.466, Z    +0.000, E1   -56.407, E3 +221162.836}
SPL {X  -160.000, Y  +554.875, Z    +0.000, E1   -61.915, E3 +221244.740}
SPL {X  -160.000, Y  +571.700, Z    +0.000, E1   -61.918, E3 +221263.817}
SPL {X  -160.000, Y  +587.975, Z    +0.000, E1   -61.909, E3 +221282.284}
SPL {X  -160.000, Y  +604.690, Z    +0.000, E1   -61.922, E3 +221301.213}
SPL {X  -160.000, Y  +621.475, Z    +0.000, E1   -61.913, E3 +221320.265}
SPL {X  -160.000, Y  +638.005, Z    +0.000, E1   -61.917, E3 +221338.995}
SPL {X  -160.000, Y  +655.083, Z    +0.000, E1   -61.921, E3 +221358.357}
SPL {X  -160.000, Y  +671.910, Z    +0.000, E1   -61.915, E3 +221377.451}
SPL {X  -159.476, Y  +687.338, Z    +0.000, E1   -61.835, E3 +221395.502}
SPL {X  -157.928, Y  +700.064, Z    +0.000, E1   -61.593, E3 +221411.567}
SPL {X  -155.236, Y  +713.154, Z    +0.000, E1   -61.225, E3 +221429.114}
SPL {X  -151.860, Y  +724.785, Z    +0.000, E1   -60.654, E3 +221445.787}
SPL {X  -148.451, Y  +734.085, Z    +0.000, E1   -60.099, E3 +221459.712}
SPL {X  -144.033, Y  +744.073, Z    +0.000, E1   -59.381, E3 +221475.232}
SPL {X  -139.170, Y  +753.341, Z    +0.000, E1   -58.489, E3 +221490.254}
SPL {X  -135.320, Y  +759.772, Z    +0.000, E1   -57.727, E3 +221500.963}
SPL {X  -117.185, Y  +783.339, Z    +0.000, E1   -48.966, E3 +221609.349}
ENDSPLINE

SPLINE
SPL {X  -142.074, Y  +747.987, Z    +0.000, E1   -38.326, E3 +221708.043}
SPL {X  -154.075, Y  +717.539, Z    +0.000, E1   -26.988, E3 +221727.200}
SPL {X  -158.904, Y  +693.092, Z    +0.000, E1   -14.171, E3 +221733.991}
SPL {X  -159.937, Y  +678.885, Z    +0.000, E1    -4.971, E3 +221735.818}
SPL {X  -160.000, Y  +672.790, Z    +0.000, E1    -0.387, E3 +221736.086}
SPL {X  -160.000, Y  +669.961, Z    +0.000, E1    +2.696, E3 +221736.163}
SPL {X  -160.000, Y  +663.591, Z    +0.000, E1   +11.688, E3 +221736.657}
SPL {X  -160.000, Y  +654.521, Z    +0.000, E1   +25.997, E3 +221738.015}
SPL {X  -160.000, Y  +642.364, Z    +0.000, E1   +40.387, E3 +221741.317}
SPL {X  -160.000, Y  +597.330, Z    +0.000, E1   +58.145, E3 +221764.228}
SPL {X  -160.000, Y  +516.293, Z    +0.000, E1   +61.751, E3 +221831.286}
SPL {X  -160.000, Y  +506.292, Z    +0.000, E1   +61.780, E3 +221842.619}
SPL {X  -160.000, Y  +494.139, Z    +0.000, E1   +61.770, E3 +221856.490}
SPL {X  -160.000, Y  +480.560, Z    +0.000, E1   +61.503, E3 +221874.287}
ENDSPLINE

SPLINE
SPL {X  -160.000, Y  +495.136, Z    +0.000, E1   +55.416, E3 +221895.793}
ENDSPLINE

SPLINE
SPL {X  -160.000, Y  +472.196, Z    +0.000, E1   +56.977, E3 +221918.468}
SPL {X  -160.000, Y  +448.172, Z    +0.000, E1   +58.434, E3 +221941.163}
SPL {X  -160.000, Y  +423.986, Z    +0.000, E1   +59.836, E3 +221962.417}
SPL {X  -160.000, Y  +398.875, Z    +0.000, E1   +61.100, E3 +221983.965}
SPL {X  -159.733, Y  +376.466, Z    +0.000, E1   +61.765, E3 +222005.154}
SPL {X  -158.128, Y  +361.299, Z    +0.000, E1   +61.520, E3 +222024.134}
SPL {X  -155.661, Y  +348.690, Z    +0.000, E1   +61.132, E3 +222041.090}
SPL {X  -152.251, Y  +336.510, Z    +0.000, E1   +60.617, E3 +222058.423}
SPL {X  -148.078, Y  +325.096, Z    +0.000, E1   +59.928, E3 +222075.551}
SPL {X  -143.290, Y  +314.510, Z    +0.000, E1   +59.129, E3 +222092.174}
SPL {X  -139.113, Y  +306.659, Z    +0.000, E1   +58.310, E3 +222105.025}
SPL {X  -135.700, Y  +300.932, Z    +0.000, E1   +57.683, E3 +222114.521}
SPL {X  -117.539, Y  +277.143, Z    +0.000, E1   +48.559, E3 +222229.207}
ENDSPLINE

SPLINE
SPL {X  -150.734, Y  +332.041, Z    +0.000, E1   +31.286, E3 +222331.872}
SPL {X  -159.235, Y  +370.077, Z    +0.000, E1   +12.240, E3 +222345.226}
SPL {X  -159.991, Y  +384.025, Z    +0.000, E1    +2.884, E3 +222346.775}
SPL {X  -160.000, Y  +388.170, Z    +0.000, E1    -0.470, E3 +222346.905}
SPL {X  -160.000, Y  +392.385, Z    +0.000, E1    -5.697, E3 +222347.096}
SPL {X  -160.000, Y  +398.918, Z    +0.000, E1   -15.420, E3 +222347.774}
SPL {X  -160.000, Y  +410.991, Z    +0.000, E1   -32.499, E3 +222350.269}
SPL {X  -160.000, Y  +455.466, Z    +0.000, E1   -56.407, E3 +222371.168}
SPL {X  -160.000, Y  +554.875, Z    +0.000, E1   -61.915, E3 +222453.072}
SPL {X  -160.000, Y  +571.700, Z    +0.000, E1   -61.918, E3 +222472.149}
SPL {X  -160.000, Y  +587.975, Z    +0.000, E1   -61.909, E3 +222490.615}
SPL {X  -160.000, Y  +604.690, Z    +0.000, E1   -61.922, E3 +222509.545}
SPL {X  -160.000, Y  +621.475, Z    +0.000, E1   -61.913, E3 +222528.597}
SPL {X  -160.000, Y  +638.005, Z    +0.000, E1   -61.917, E3 +222547.327}
SPL {X  -160.000, Y  +655.083, Z    +0.000, E1   -61.921, E3 +222566.688}
SPL {X  -160.000, Y  +671.910, Z    +0.000, E1   -61.915, E3 +222585.782}
SPL {X  -159.476, Y  +687.338, Z    +0.000, E1   -61.835, E3 +222603.834}
SPL {X  -157.928, Y  +700.064, Z    +0.000, E1   -61.593, E3 +222619.899}
SPL {X  -155.236, Y  +713.154, Z    +0.000, E1   -61.225, E3 +222637.446}
SPL {X  -151.860, Y  +724.785, Z    +0.000, E1   -60.654, E3 +222654.118}
SPL {X  -148.451, Y  +734.085, Z    +0.000, E1   -60.099, E3 +222668.044}
SPL {X  -144.033, Y  +744.073, Z    +0.000, E1   -59.381, E3 +222683.564}
SPL {X  -139.170, Y  +753.341, Z    +0.000, E1   -58.489, E3 +222698.585}
SPL {X  -135.320, Y  +759.772, Z    +0.000, E1   -57.727, E3 +222709.295}
SPL {X  -117.185, Y  +783.339, Z    +0.000, E1   -48.966, E3 +222817.681}
ENDSPLINE

SPLINE
SPL {X  -142.074, Y  +747.987, Z    +0.000, E1   -38.326, E3 +222916.375}
SPL {X  -154.075, Y  +717.539, Z    +0.000, E1   -26.988, E3 +222935.532}
SPL {X  -158.904, Y  +693.092, Z    +0.000, E1   -14.171, E3 +222942.323}
SPL {X  -159.937, Y  +678.885, Z    +0.000, E1    -4.971, E3 +222944.150}
SPL {X  -160.000, Y  +672.790, Z    +0.000, E1    -0.387, E3 +222944.418}
SPL {X  -160.000, Y  +669.961, Z    +0.000, E1    +2.696, E3 +222944.495}
SPL {X  -160.000, Y  +663.591, Z    +0.000, E1   +11.688, E3 +222944.989}
SPL {X  -160.000, Y  +654.521, Z    +0.000, E1   +25.997, E3 +222946.347}
SPL {X  -160.000, Y  +642.364, Z    +0.000, E1   +40.387, E3 +222949.649}
SPL {X  -160.000, Y  +597.330, Z    +0.000, E1   +58.145, E3 +222972.560}
SPL {X  -160.000, Y  +516.293, Z    +0.000, E1   +61.751, E3 +223039.617}
SPL {X  -160.000, Y  +506.292, Z    +0.000, E1   +61.780, E3 +223050.951}
SPL {X  -160.000, Y  +494.139, Z    +0.000, E1   +61.770, E3 +223064.821}
SPL {X  -160.000, Y  +480.560, Z    +0.000, E1   +61.503, E3 +223082.618}
ENDSPLINE

SPLINE
SPL {X  -160.000, Y  +495.136, Z    +0.000, E1   +55.416, E3 +223104.125}
ENDSPLINE

SPLINE
SPL {X  -160.000, Y  +472.196, Z    +0.000, E1   +56.977, E3 +223126.800}
SPL {X  -160.000, Y  +448.172, Z    +0.000, E1   +58.434, E3 +223149.495}
SPL {X  -160.000, Y  +423.986, Z    +0.000, E1   +59.836, E3 +223170.748}
SPL {X  -160.000, Y  +398.875, Z    +0.000, E1   +61.100, E3 +223192.296}
SPL {X  -159.733, Y  +376.466, Z    +0.000, E1   +61.765, E3 +223213.486}
SPL {X  -158.128, Y  +361.299, Z    +0.000, E1   +61.520, E3 +223232.465}
SPL {X  -155.661, Y  +348.690, Z    +0.000, E1   +61.132, E3 +223249.422}
SPL {X  -152.251, Y  +336.510, Z    +0.000, E1   +60.617, E3 +223266.754}
SPL {X  -148.078, Y  +325.096, Z    +0.000, E1   +59.928, E3 +223283.883}
SPL {X  -143.290, Y  +314.510, Z    +0.000, E1   +59.129, E3 +223300.506}
SPL {X  -139.113, Y  +306.659, Z    +0.000, E1   +58.310, E3 +223313.356}
SPL {X  -135.700, Y  +300.932, Z    +0.000, E1   +57.683, E3 +223322.853}
SPL {X  -117.539, Y  +277.143, Z    +0.000, E1   +48.559, E3 +223437.539}
ENDSPLINE

SPLINE
SPL {X  -150.734, Y  +332.041, Z    +0.000, E1   +31.286, E3 +223540.204}
SPL {X  -159.235, Y  +370.077, Z    +0.000, E1   +12.240, E3 +223553.558}
SPL {X  -159.991, Y  +384.025, Z    +0.000, E1    +2.884, E3 +223555.107}
SPL {X  -160.000, Y  +388.170, Z    +0.000, E1    -0.470, E3 +223555.237}
SPL {X  -160.000, Y  +392.385, Z    +0.000, E1    -5.697, E3 +223555.427}
SPL {X  -160.000, Y  +398.918, Z    +0.000, E1   -15.420, E3 +223556.106}
SPL {X  -160.000, Y  +410.991, Z    +0.000, E1   -32.499, E3 +223558.601}
SPL {X  -160.000, Y  +455.466, Z    +0.000, E1   -56.407, E3 +223579.500}
SPL {X  -160.000, Y  +554.875, Z    +0.000, E1   -61.915, E3 +223661.404}
SPL {X  -160.000, Y  +571.700, Z    +0.000, E1   -61.918, E3 +223680.481}
SPL {X  -160.000, Y  +587.975, Z    +0.000, E1   -61.909, E3 +223698.947}
SPL {X  -160.000, Y  +604.690, Z    +0.000, E1   -61.922, E3 +223717.876}
SPL {X  -160.000, Y  +621.475, Z    +0.000, E1   -61.913, E3 +223736.928}
SPL {X  -160.000, Y  +638.005, Z    +0.000, E1   -61.917, E3 +223755.659}
SPL {X  -160.000, Y  +655.083, Z    +0.000, E1   -61.921, E3 +223775.020}
SPL {X  -160.000, Y  +671.910, Z    +0.000, E1   -61.915, E3 +223794.114}
SPL {X  -159.476, Y  +687.338, Z    +0.000, E1   -61.835, E3 +223812.166}
SPL {X  -157.928, Y  +700.064, Z    +0.000, E1   -61.593, E3 +223828.230}
SPL {X  -155.236, Y  +713.154, Z    +0.000, E1   -61.225, E3 +223845.778}
SPL {X  -151.860, Y  +724.785, Z    +0.000, E1   -60.654, E3 +223862.450}
SPL {X  -148.451, Y  +734.085, Z    +0.000, E1   -60.099, E3 +223876.375}
SPL {X  -144.033, Y  +744.073, Z    +0.000, E1   -59.381, E3 +223891.896}
SPL {X  -139.170, Y  +753.341, Z    +0.000, E1   -58.489, E3 +223906.917}
SPL {X  -135.320, Y  +759.772, Z    +0.000, E1   -57.727, E3 +223917.627}
SPL {X  -117.185, Y  +783.339, Z    +0.000, E1   -48.966, E3 +224026.013}
ENDSPLINE

SPLINE
SPL {X  -142.074, Y  +747.987, Z    +0.000, E1   -38.326, E3 +224124.707}
SPL {X  -154.075, Y  +717.539, Z    +0.000, E1   -26.988, E3 +224143.864}
SPL {X  -158.904, Y  +693.092, Z    +0.000, E1   -14.171, E3 +224150.655}
SPL {X  -159.937, Y  +678.885, Z    +0.000, E1    -4.971, E3 +224152.482}
SPL {X  -160.000, Y  +672.790, Z    +0.000, E1    -0.387, E3 +224152.750}
SPL {X  -160.000, Y  +669.961, Z    +0.000, E1    +2.696, E3 +224152.826}
SPL {X  -160.000, Y  +663.591, Z    +0.000, E1   +11.688, E3 +224153.321}
SPL {X  -160.000, Y  +654.521, Z    +0.000, E1   +25.997, E3 +224154.679}
SPL {X  -160.000, Y  +642.364, Z    +0.000, E1   +40.387, E3 +224157.981}
SPL {X  -160.000, Y  +597.330, Z    +0.000, E1   +58.145, E3 +224180.892}
SPL {X  -160.000, Y  +516.293, Z    +0.000, E1   +61.751, E3 +224247.949}
SPL {X  -160.000, Y  +506.292, Z    +0.000, E1   +61.780, E3 +224259.283}
SPL {X  -160.000, Y  +494.139, Z    +0.000, E1   +61.770, E3 +224273.153}
SPL {X  -160.000, Y  +480.560, Z    +0.000, E1   +61.503, E3 +224290.950}
ENDSPLINE

SPLINE
SPL {X  -160.000, Y  +495.136, Z    +0.000, E1   +55.416, E3 +224312.457}
ENDSPLINE

SPLINE
SPL {X  -160.000, Y  +472.196, Z    +0.000, E1   +56.977, E3 +224335.132}
SPL {X  -160.000, Y  +448.172, Z    +0.000, E1   +58.434, E3 +224357.826}
SPL {X  -160.000, Y  +423.986, Z    +0.000, E1   +59.836, E3 +224379.080}
SPL {X  -160.000, Y  +398.875, Z    +0.000, E1   +61.100, E3 +224400.628}
SPL {X  -159.733, Y  +376.466, Z    +0.000, E1   +61.765, E3 +224421.818}
SPL {X  -158.128, Y  +361.299, Z    +0.000, E1   +61.520, E3 +224440.797}
SPL {X  -155.661, Y  +348.690, Z    +0.000, E1   +61.132, E3 +224457.753}
SPL {X  -152.251, Y  +336.510, Z    +0.000, E1   +60.617, E3 +224475.086}
SPL {X  -148.078, Y  +325.096, Z    +0.000, E1   +59.928, E3 +224492.215}
SPL {X  -143.290, Y  +314.510, Z    +0.000, E1   +59.129, E3 +224508.837}
SPL {X  -139.113, Y  +306.659, Z    +0.000, E1   +58.310, E3 +224521.688}
SPL {X  -135.700, Y  +300.932, Z    +0.000, E1   +57.683, E3 +224531.185}
SPL {X  -117.539, Y  +277.143, Z    +0.000, E1   +48.559, E3 +224645.871}
ENDSPLINE

SPLINE
SPL {X  -150.734, Y  +332.041, Z    +0.000, E1   +31.286, E3 +224748.535}
SPL {X  -159.235, Y  +370.077, Z    +0.000, E1   +12.240, E3 +224761.890}
SPL {X  -159.991, Y  +384.025, Z    +0.000, E1    +2.884, E3 +224763.438}
SPL {X  -160.000, Y  +388.170, Z    +0.000, E1    -0.470, E3 +224763.569}
SPL {X  -160.000, Y  +392.385, Z    +0.000, E1    -5.697, E3 +224763.759}
SPL {X  -160.000, Y  +398.918, Z    +0.000, E1   -15.420, E3 +224764.438}
SPL {X  -160.000, Y  +410.991, Z    +0.000, E1   -32.499, E3 +224766.933}
SPL {X  -160.000, Y  +455.466, Z    +0.000, E1   -56.407, E3 +224787.832}
SPL {X  -160.000, Y  +554.875, Z    +0.000, E1   -61.915, E3 +224869.736}
SPL {X  -160.000, Y  +571.700, Z    +0.000, E1   -61.918, E3 +224888.812}
SPL {X  -160.000, Y  +587.975, Z    +0.000, E1   -61.909, E3 +224907.279}
SPL {X  -160.000, Y  +604.690, Z    +0.000, E1   -61.922, E3 +224926.208}
SPL {X  -160.000, Y  +621.475, Z    +0.000, E1   -61.913, E3 +224945.260}
SPL {X  -160.000, Y  +638.005, Z    +0.000, E1   -61.917, E3 +224963.990}
SPL {X  -160.000, Y  +655.083, Z    +0.000, E1   -61.921, E3 +224983.352}
SPL {X  -160.000, Y  +671.910, Z    +0.000, E1   -61.915, E3 +225002.446}
SPL {X  -159.476, Y  +687.338, Z    +0.000, E1   -61.835, E3 +225020.498}
SPL {X  -157.928, Y  +700.064, Z    +0.000, E1   -61.593, E3 +225036.562}
SPL {X  -155.236, Y  +713.154, Z    +0.000, E1   -61.225, E3 +225054.109}
SPL {X  -151.860, Y  +724.785, Z    +0.000, E1   -60.654, E3 +225070.782}
SPL {X  -148.451, Y  +734.085, Z    +0.000, E1   -60.099, E3 +225084.707}
SPL {X  -144.033, Y  +744.073, Z    +0.000, E1   -59.381, E3 +225100.227}
SPL {X  -139.170, Y  +753.341, Z    +0.000, E1   -58.489, E3 +225115.249}
SPL {X  -135.320, Y  +759.772, Z    +0.000, E1   -57.727, E3 +225125.958}
SPL {X  -117.014, Y  +783.523, Z    +0.000, E1   -50.796, E3 +225209.004}
ENDSPLINE

SPLINE
SPL {X  -117.768, Y  +782.709, Z    +0.000, E1   -48.245, E3 +225244.683}
SPL {X  -142.074, Y  +747.987, Z    +0.000, E1   -38.326, E3 +225333.038}
SPL {X  -154.075, Y  +717.539, Z    +0.000, E1   -26.988, E3 +225352.195}
SPL {X  -158.904, Y  +693.092, Z    +0.000, E1   -14.171, E3 +225358.986}
SPL {X  -159.937, Y  +678.885, Z    +0.000, E1    -4.971, E3 +225360.814}
SPL {X  -160.000, Y  +672.790, Z    +0.000, E1    -0.387, E3 +225361.081}
SPL {X  -160.000, Y  +669.961, Z    +0.000, E1    +2.696, E3 +225361.158}
SPL {X  -160.000, Y  +663.591, Z    +0.000, E1   +11.688, E3 +225361.652}
SPL {X  -160.000, Y  +654.521, Z    +0.000, E1   +25.997, E3 +225363.010}
SPL {X  -160.000, Y  +642.364, Z    +0.000, E1   +40.387, E3 +225366.312}
SPL {X  -160.000, Y  +597.330, Z    +0.000, E1   +58.145, E3 +225389.224}
SPL {X  -160.000, Y  +516.293, Z    +0.000, E1   +61.751, E3 +225456.281}
SPL {X  -160.000, Y  +506.292, Z    +0.000, E1   +61.780, E3 +225467.615}
SPL {X  -160.000, Y  +494.139, Z    +0.000, E1   +61.770, E3 +225481.485}
SPL {X  -160.000, Y  +480.560, Z    +0.000, E1   +61.503, E3 +225499.282}
ENDSPLINE

SPLINE
SPL {X  -160.000, Y  +495.136, Z    +0.000, E1   +55.416, E3 +225520.789}
ENDSPLINE

SPLINE
SPL {X  -160.000, Y  +472.196, Z    +0.000, E1   +56.977, E3 +225543.463}
SPL {X  -160.000, Y  +448.172, Z    +0.000, E1   +58.434, E3 +225566.158}
SPL {X  -160.000, Y  +423.986, Z    +0.000, E1   +59.836, E3 +225587.412}
SPL {X  -160.000, Y  +398.875, Z    +0.000, E1   +61.100, E3 +225608.960}
ENDSPLINE

SPLINE
SPL {X  -160.000, Y  +391.117, Z    +0.000, E1   +59.361, E3 +225630.320}
SPL {X  -159.620, Y  +374.678, Z    +0.000, E1   +59.299, E3 +225651.443}
SPL {X  -157.749, Y  +358.956, Z    +0.000, E1   +59.037, E3 +225673.141}
SPL {X  -154.809, Y  +345.275, Z    +0.000, E1   +58.527, E3 +225693.465}
SPL {X  -151.181, Y  +333.313, Z    +0.000, E1   +57.939, E3 +225712.173}
SPL {X  -146.730, Y  +321.901, Z    +0.000, E1   +57.169, E3 +225730.919}
SPL {X  -142.568, Y  +313.075, Z    +0.000, E1   +56.366, E3 +225746.040}
SPL {X  -138.721, Y  +305.972, Z    +0.000, E1   +55.652, E3 +225758.468}
SPL {X  -123.439, Y  +283.902, Z    +0.000, E1   +48.158, E3 +225849.993}
ENDSPLINE

SPLINE
SPL {X  -141.803, Y  +311.593, Z    +0.000, E1   +37.608, E3 +225940.612}
SPL {X  -154.548, Y  +344.290, Z    +0.000, E1   +25.264, E3 +225965.095}
SPL {X  -159.249, Y  +370.212, Z    +0.000, E1   +11.801, E3 +225973.128}
SPL {X  -159.987, Y  +383.623, Z    +0.000, E1    +3.169, E3 +225974.881}
SPL {X  -160.000, Y  +388.238, Z    +0.000, E1    -0.420, E3 +225975.092}
SPL {X  -160.000, Y  +392.418, Z    +0.000, E1    -5.131, E3 +225975.332}
SPL {X  -160.000, Y  +399.157, Z    +0.000, E1   -14.351, E3 +225976.149}
SPL {X  -160.000, Y  +411.277, Z    +0.000, E1   -30.487, E3 +225978.927}
SPL {X  -160.000, Y  +452.990, Z    +0.000, E1   -53.470, E3 +226000.291}
SPL {X  -160.000, Y  +539.177, Z    +0.000, E1   -59.280, E3 +226078.617}
SPL {X  -160.000, Y  +554.731, Z    +0.000, E1   -59.281, E3 +226098.262}
SPL {X  -160.000, Y  +572.172, Z    +0.000, E1   -59.312, E3 +226120.225}
SPL {X  -160.000, Y  +589.502, Z    +0.000, E1   -59.284, E3 +226142.163}
SPL {X  -160.000, Y  +604.577, Z    +0.000, E1   -59.272, E3 +226161.222}
SPL {X  -160.000, Y  +620.386, Z    +0.000, E1   -59.294, E3 +226181.149}
SPL {X  -160.000, Y  +636.664, Z    +0.000, E1   -59.282, E3 +226201.739}
SPL {X  -160.000, Y  +654.257, Z    +0.000, E1   -59.312, E3 +226223.917}
SPL {X  -160.000, Y  +671.385, Z    +0.000, E1   -59.278, E3 +226245.606}
SPL {X  -159.497, Y  +687.081, Z    +0.000, E1   -59.218, E3 +226265.934}
SPL {X  -157.563, Y  +702.220, Z    +0.000, E1   -58.916, E3 +226287.095}
SPL {X  -154.922, Y  +714.390, Z    +0.000, E1   -58.446, E3 +226305.289}
SPL {X  -151.559, Y  +725.681, Z    +0.000, E1   -57.922, E3 +226322.919}
SPL {X  -147.777, Y  +735.736, Z    +0.000, E1   -57.226, E3 +226339.414}
SPL {X  -143.698, Y  +744.763, Z    +0.000, E1   -56.526, E3 +226354.690}
SPL {X  -138.992, Y  +753.654, Z    +0.000, E1   -55.630, E3 +226370.268}
SPL {X  -122.847, Y  +776.912, Z    +0.000, E1   -47.251, E3 +226479.950}
ENDSPLINE

SPLINE
SPL {X  -149.319, Y  +731.879, Z    +0.000, E1   -32.249, E3 +226574.337}
SPL {X  -158.304, Y  +697.637, Z    +0.000, E1   -16.440, E3 +226588.988}
SPL {X  -159.863, Y  +681.030, Z    +0.000, E1    -6.312, E3 +226591.930}
SPL {X  -160.000, Y  +673.530, Z    +0.000, E1    -1.059, E3 +226592.437}
SPL {X  -160.000, Y  +670.245, Z    +0.000, E1    +2.042, E3 +226592.550}
SPL {X  -160.000, Y  +663.790, Z    +0.000, E1   +10.467, E3 +226593.074}
SPL {X  -160.000, Y  +655.457, Z    +0.000, E1   +22.866, E3 +226594.437}
SPL {X  -160.000, Y  +644.540, Z    +0.000, E1   +36.054, E3 +226597.468}
SPL {X  -160.000, Y  +601.495, Z    +0.000, E1   +56.174, E3 +226618.397}
SPL {X  -160.000, Y  +515.545, Z    +0.000, E1   +60.629, E3 +226693.791}
SPL {X  -160.000, Y  +503.330, Z    +0.000, E1   +60.630, E3 +226708.397}
SPL {X  -160.000, Y  +487.139, Z    +0.000, E1   +60.676, E3 +226727.665}
SPL {X  -160.000, Y  +466.770, Z    +0.000, E1   +60.698, E3 +226751.960}
SPL {X  -160.000, Y  +454.269, Z    +0.000, E1   +59.898, E3 +226772.211}
ENDSPLINE

SPLINE
SPL {X  -160.000, Y  +458.973, Z    +0.000, E1   +55.880, E3 +226793.130}
ENDSPLINE

SPLINE
SPL {X  -160.000, Y  +435.816, Z    +0.000, E1   +57.237, E3 +226816.805}
SPL {X  -160.000, Y  +411.824, Z    +0.000, E1   +58.675, E3 +226839.299}
SPL {X  -160.000, Y  +390.940, Z    +0.000, E1   +59.356, E3 +226861.327}
SPL {X  -159.620, Y  +374.678, Z    +0.000, E1   +59.299, E3 +226882.211}
SPL {X  -157.749, Y  +358.956, Z    +0.000, E1   +59.037, E3 +226903.909}
SPL {X  -154.809, Y  +345.275, Z    +0.000, E1   +58.527, E3 +226924.232}
SPL {X  -151.181, Y  +333.313, Z    +0.000, E1   +57.939, E3 +226942.940}
SPL {X  -146.730, Y  +321.901, Z    +0.000, E1   +57.169, E3 +226961.686}
SPL {X  -142.568, Y  +313.075, Z    +0.000, E1   +56.366, E3 +226976.808}
SPL {X  -139.172, Y  +306.763, Z    +0.000, E1   +55.717, E3 +226987.862}
SPL {X  -137.037, Y  +303.112, Z    +0.000, E1   +55.261, E3 +226994.409}
SPL {X  -123.439, Y  +283.902, Z    +0.000, E1   +48.158, E3 +227080.760}
ENDSPLINE

SPLINE
SPL {X  -141.803, Y  +311.593, Z    +0.000, E1   +37.608, E3 +227171.379}
SPL {X  -154.548, Y  +344.290, Z    +0.000, E1   +25.264, E3 +227195.863}
SPL {X  -159.249, Y  +370.212, Z    +0.000, E1   +11.801, E3 +227203.895}
SPL {X  -159.987, Y  +383.623, Z    +0.000, E1    +3.169, E3 +227205.648}
SPL {X  -160.000, Y  +388.238, Z    +0.000, E1    -0.420, E3 +227205.859}
SPL {X  -160.000, Y  +392.418, Z    +0.000, E1    -5.131, E3 +227206.100}
SPL {X  -160.000, Y  +399.157, Z    +0.000, E1   -14.351, E3 +227206.916}
SPL {X  -160.000, Y  +411.277, Z    +0.000, E1   -30.487, E3 +227209.694}
SPL {X  -160.000, Y  +452.990, Z    +0.000, E1   -53.470, E3 +227231.058}
SPL {X  -160.000, Y  +539.177, Z    +0.000, E1   -59.280, E3 +227309.385}
SPL {X  -160.000, Y  +554.731, Z    +0.000, E1   -59.281, E3 +227329.029}
SPL {X  -160.000, Y  +572.172, Z    +0.000, E1   -59.312, E3 +227350.992}
SPL {X  -160.000, Y  +589.502, Z    +0.000, E1   -59.284, E3 +227372.930}
SPL {X  -160.000, Y  +604.577, Z    +0.000, E1   -59.272, E3 +227391.989}
SPL {X  -160.000, Y  +620.386, Z    +0.000, E1   -59.294, E3 +227411.917}
SPL {X  -160.000, Y  +636.664, Z    +0.000, E1   -59.282, E3 +227432.506}
SPL {X  -160.000, Y  +654.257, Z    +0.000, E1   -59.312, E3 +227454.685}
SPL {X  -160.000, Y  +671.385, Z    +0.000, E1   -59.278, E3 +227476.374}
SPL {X  -159.497, Y  +687.081, Z    +0.000, E1   -59.218, E3 +227496.701}
SPL {X  -157.563, Y  +702.220, Z    +0.000, E1   -58.916, E3 +227517.862}
SPL {X  -154.922, Y  +714.390, Z    +0.000, E1   -58.446, E3 +227536.056}
SPL {X  -151.559, Y  +725.681, Z    +0.000, E1   -57.922, E3 +227553.687}
SPL {X  -147.777, Y  +735.736, Z    +0.000, E1   -57.226, E3 +227570.181}
SPL {X  -143.698, Y  +744.763, Z    +0.000, E1   -56.526, E3 +227585.458}
SPL {X  -138.992, Y  +753.654, Z    +0.000, E1   -55.630, E3 +227601.035}
SPL {X  -122.847, Y  +776.912, Z    +0.000, E1   -47.251, E3 +227710.718}
ENDSPLINE

SPLINE
SPL {X  -149.319, Y  +731.879, Z    +0.000, E1   -32.249, E3 +227805.104}
SPL {X  -158.304, Y  +697.637, Z    +0.000, E1   -16.440, E3 +227819.755}
SPL {X  -159.863, Y  +681.030, Z    +0.000, E1    -6.312, E3 +227822.697}
SPL {X  -160.000, Y  +673.530, Z    +0.000, E1    -1.059, E3 +227823.204}
SPL {X  -160.000, Y  +670.245, Z    +0.000, E1    +2.042, E3 +227823.317}
SPL {X  -160.000, Y  +663.790, Z    +0.000, E1   +10.467, E3 +227823.842}
SPL {X  -160.000, Y  +655.457, Z    +0.000, E1   +22.866, E3 +227825.204}
SPL {X  -160.000, Y  +644.540, Z    +0.000, E1   +36.054, E3 +227828.235}
SPL {X  -160.000, Y  +601.495, Z    +0.000, E1   +56.174, E3 +227849.164}
SPL {X  -160.000, Y  +515.545, Z    +0.000, E1   +60.629, E3 +227924.558}
SPL {X  -160.000, Y  +503.330, Z    +0.000, E1   +60.630, E3 +227939.164}
SPL {X  -160.000, Y  +487.139, Z    +0.000, E1   +60.676, E3 +227958.432}
SPL {X  -160.000, Y  +466.770, Z    +0.000, E1   +60.698, E3 +227982.728}
SPL {X  -160.000, Y  +454.269, Z    +0.000, E1   +59.898, E3 +228002.979}
ENDSPLINE

SPLINE
SPL {X  -160.000, Y  +458.973, Z    +0.000, E1   +55.880, E3 +228023.897}
ENDSPLINE

SPLINE
SPL {X  -160.000, Y  +435.816, Z    +0.000, E1   +57.237, E3 +228047.573}
SPL {X  -160.000, Y  +411.824, Z    +0.000, E1   +58.675, E3 +228070.066}
SPL {X  -160.000, Y  +390.940, Z    +0.000, E1   +59.356, E3 +228092.094}
SPL {X  -159.620, Y  +374.678, Z    +0.000, E1   +59.299, E3 +228112.978}
SPL {X  -157.749, Y  +358.956, Z    +0.000, E1   +59.037, E3 +228134.676}
SPL {X  -154.809, Y  +345.275, Z    +0.000, E1   +58.527, E3 +228154.999}
SPL {X  -151.181, Y  +333.313, Z    +0.000, E1   +57.939, E3 +228173.708}
SPL {X  -146.730, Y  +321.901, Z    +0.000, E1   +57.169, E3 +228192.453}
SPL {X  -142.568, Y  +313.075, Z    +0.000, E1   +56.366, E3 +228207.575}
SPL {X  -138.721, Y  +305.972, Z    +0.000, E1   +55.652, E3 +228220.003}
SPL {X  -123.439, Y  +283.902, Z    +0.000, E1   +48.158, E3 +228311.527}
ENDSPLINE

SPLINE
SPL {X  -141.803, Y  +311.593, Z    +0.000, E1   +37.608, E3 +228402.147}
SPL {X  -154.548, Y  +344.290, Z    +0.000, E1   +25.264, E3 +228426.630}
SPL {X  -159.249, Y  +370.212, Z    +0.000, E1   +11.801, E3 +228434.662}
SPL {X  -159.987, Y  +383.623, Z    +0.000, E1    +3.169, E3 +228436.415}
SPL {X  -160.000, Y  +388.238, Z    +0.000, E1    -0.420, E3 +228436.627}
SPL {X  -160.000, Y  +392.418, Z    +0.000, E1    -5.131, E3 +228436.867}
SPL {X  -160.000, Y  +399.157, Z    +0.000, E1   -14.351, E3 +228437.683}
SPL {X  -160.000, Y  +411.277, Z    +0.000, E1   -30.487, E3 +228440.461}
SPL {X  -160.000, Y  +452.990, Z    +0.000, E1   -53.470, E3 +228461.825}
SPL {X  -160.000, Y  +539.177, Z    +0.000, E1   -59.280, E3 +228540.152}
SPL {X  -160.000, Y  +554.731, Z    +0.000, E1   -59.281, E3 +228559.796}
SPL {X  -160.000, Y  +572.172, Z    +0.000, E1   -59.312, E3 +228581.759}
SPL {X  -160.000, Y  +589.502, Z    +0.000, E1   -59.284, E3 +228603.697}
SPL {X  -160.000, Y  +604.577, Z    +0.000, E1   -59.272, E3 +228622.757}
SPL {X  -160.000, Y  +620.386, Z    +0.000, E1   -59.294, E3 +228642.684}
SPL {X  -160.000, Y  +636.664, Z    +0.000, E1   -59.282, E3 +228663.274}
SPL {X  -160.000, Y  +654.257, Z    +0.000, E1   -59.312, E3 +228685.452}
SPL {X  -160.000, Y  +671.385, Z    +0.000, E1   -59.278, E3 +228707.141}
SPL {X  -159.497, Y  +687.081, Z    +0.000, E1   -59.218, E3 +228727.468}
SPL {X  -157.563, Y  +702.220, Z    +0.000, E1   -58.916, E3 +228748.630}
SPL {X  -154.922, Y  +714.390, Z    +0.000, E1   -58.446, E3 +228766.823}
SPL {X  -151.559, Y  +725.681, Z    +0.000, E1   -57.922, E3 +228784.454}
SPL {X  -147.777, Y  +735.736, Z    +0.000, E1   -57.226, E3 +228800.948}
SPL {X  -143.698, Y  +744.763, Z    +0.000, E1   -56.526, E3 +228816.225}
SPL {X  -138.992, Y  +753.654, Z    +0.000, E1   -55.630, E3 +228831.802}
SPL {X  -122.847, Y  +776.912, Z    +0.000, E1   -47.251, E3 +228941.485}
ENDSPLINE

SPLINE
SPL {X  -149.319, Y  +731.879, Z    +0.000, E1   -32.249, E3 +229035.872}
SPL {X  -158.304, Y  +697.637, Z    +0.000, E1   -16.440, E3 +229050.522}
SPL {X  -159.863, Y  +681.030, Z    +0.000, E1    -6.312, E3 +229053.464}
SPL {X  -160.000, Y  +673.530, Z    +0.000, E1    -1.059, E3 +229053.971}
SPL {X  -160.000, Y  +670.245, Z    +0.000, E1    +2.042, E3 +229054.084}
SPL {X  -160.000, Y  +663.790, Z    +0.000, E1   +10.467, E3 +229054.609}
SPL {X  -160.000, Y  +655.457, Z    +0.000, E1   +22.866, E3 +229055.971}
SPL {X  -160.000, Y  +644.540, Z    +0.000, E1   +36.054, E3 +229059.002}
SPL {X  -160.000, Y  +601.495, Z    +0.000, E1   +56.174, E3 +229079.931}
SPL {X  -160.000, Y  +515.545, Z    +0.000, E1   +60.629, E3 +229155.325}
SPL {X  -160.000, Y  +503.330, Z    +0.000, E1   +60.630, E3 +229169.931}
SPL {X  -160.000, Y  +487.139, Z    +0.000, E1   +60.676, E3 +229189.199}
SPL {X  -160.000, Y  +466.770, Z    +0.000, E1   +60.698, E3 +229213.495}
SPL {X  -160.000, Y  +454.269, Z    +0.000, E1   +59.898, E3 +229233.746}
ENDSPLINE

SPLINE
SPL {X  -160.000, Y  +458.973, Z    +0.000, E1   +55.880, E3 +229254.664}
ENDSPLINE

SPLINE
SPL {X  -160.000, Y  +435.816, Z    +0.000, E1   +57.237, E3 +229278.340}
SPL {X  -160.000, Y  +411.824, Z    +0.000, E1   +58.675, E3 +229300.834}
SPL {X  -160.000, Y  +390.940, Z    +0.000, E1   +59.356, E3 +229322.861}
SPL {X  -159.620, Y  +374.678, Z    +0.000, E1   +59.299, E3 +229343.745}
SPL {X  -157.749, Y  +358.956, Z    +0.000, E1   +59.037, E3 +229365.443}
SPL {X  -154.809, Y  +345.275, Z    +0.000, E1   +58.527, E3 +229385.766}
SPL {X  -151.181, Y  +333.313, Z    +0.000, E1   +57.939, E3 +229404.475}
SPL {X  -146.730, Y  +321.901, Z    +0.000, E1   +57.169, E3 +229423.220}
SPL {X  -142.568, Y  +313.075, Z    +0.000, E1   +56.366, E3 +229438.342}
SPL {X  -139.172, Y  +306.763, Z    +0.000, E1   +55.717, E3 +229449.397}
SPL {X  -137.037, Y  +303.112, Z    +0.000, E1   +55.261, E3 +229455.943}
SPL {X  -123.439, Y  +283.902, Z    +0.000, E1   +48.158, E3 +229542.295}
ENDSPLINE

SPLINE
SPL {X  -141.803, Y  +311.593, Z    +0.000, E1   +37.608, E3 +229632.914}
SPL {X  -154.548, Y  +344.290, Z    +0.000, E1   +25.264, E3 +229657.397}
SPL {X  -159.249, Y  +370.212, Z    +0.000, E1   +11.801, E3 +229665.429}
SPL {X  -159.987, Y  +383.623, Z    +0.000, E1    +3.169, E3 +229667.182}
SPL {X  -160.000, Y  +388.238, Z    +0.000, E1    -0.420, E3 +229667.394}
SPL {X  -160.000, Y  +392.418, Z    +0.000, E1    -5.131, E3 +229667.634}
SPL {X  -160.000, Y  +399.157, Z    +0.000, E1   -14.351, E3 +229668.451}
SPL {X  -160.000, Y  +411.277, Z    +0.000, E1   -30.487, E3 +229671.229}
SPL {X  -160.000, Y  +452.990, Z    +0.000, E1   -53.470, E3 +229692.593}
SPL {X  -160.000, Y  +539.177, Z    +0.000, E1   -59.280, E3 +229770.919}
SPL {X  -160.000, Y  +554.731, Z    +0.000, E1   -59.281, E3 +229790.564}
SPL {X  -160.000, Y  +572.172, Z    +0.000, E1   -59.312, E3 +229812.526}
SPL {X  -160.000, Y  +589.502, Z    +0.000, E1   -59.284, E3 +229834.465}
SPL {X  -160.000, Y  +604.577, Z    +0.000, E1   -59.272, E3 +229853.524}
SPL {X  -160.000, Y  +620.386, Z    +0.000, E1   -59.294, E3 +229873.451}
SPL {X  -160.000, Y  +636.664, Z    +0.000, E1   -59.282, E3 +229894.041}
SPL {X  -160.000, Y  +654.257, Z    +0.000, E1   -59.312, E3 +229916.219}
SPL {X  -160.000, Y  +671.385, Z    +0.000, E1   -59.278, E3 +229937.908}
SPL {X  -159.497, Y  +687.081, Z    +0.000, E1   -59.218, E3 +229958.235}
SPL {X  -157.563, Y  +702.220, Z    +0.000, E1   -58.916, E3 +229979.397}
SPL {X  -154.922, Y  +714.390, Z    +0.000, E1   -58.446, E3 +229997.590}
SPL {X  -151.559, Y  +725.681, Z    +0.000, E1   -57.922, E3 +230015.221}
SPL {X  -147.777, Y  +735.736, Z    +0.000, E1   -57.226, E3 +230031.716}
SPL {X  -143.698, Y  +744.763, Z    +0.000, E1   -56.526, E3 +230046.992}
SPL {X  -138.992, Y  +753.654, Z    +0.000, E1   -55.630, E3 +230062.569}
SPL {X  -122.847, Y  +776.912, Z    +0.000, E1   -47.251, E3 +230172.252}
ENDSPLINE

SPLINE
SPL {X  -149.319, Y  +731.879, Z    +0.000, E1   -32.249, E3 +230266.639}
SPL {X  -158.304, Y  +697.637, Z    +0.000, E1   -16.440, E3 +230281.289}
SPL {X  -159.863, Y  +681.030, Z    +0.000, E1    -6.312, E3 +230284.232}
SPL {X  -160.000, Y  +673.530, Z    +0.000, E1    -1.059, E3 +230284.738}
SPL {X  -160.000, Y  +670.245, Z    +0.000, E1    +2.042, E3 +230284.852}
SPL {X  -160.000, Y  +663.790, Z    +0.000, E1   +10.467, E3 +230285.376}
SPL {X  -160.000, Y  +655.457, Z    +0.000, E1   +22.866, E3 +230286.738}
SPL {X  -160.000, Y  +644.540, Z    +0.000, E1   +36.054, E3 +230289.769}
SPL {X  -160.000, Y  +601.495, Z    +0.000, E1   +56.174, E3 +230310.699}
SPL {X  -160.000, Y  +515.545, Z    +0.000, E1   +60.629, E3 +230386.093}
SPL {X  -160.000, Y  +503.330, Z    +0.000, E1   +60.630, E3 +230400.698}
SPL {X  -160.000, Y  +487.139, Z    +0.000, E1   +60.676, E3 +230419.967}
SPL {X  -160.000, Y  +466.770, Z    +0.000, E1   +60.698, E3 +230444.262}
SPL {X  -160.000, Y  +454.269, Z    +0.000, E1   +59.898, E3 +230464.513}
ENDSPLINE

SPLINE
SPL {X  -160.000, Y  +458.973, Z    +0.000, E1   +55.880, E3 +230485.432}
ENDSPLINE

SPLINE
SPL {X  -160.000, Y  +435.816, Z    +0.000, E1   +57.237, E3 +230509.107}
SPL {X  -160.000, Y  +411.824, Z    +0.000, E1   +58.675, E3 +230531.601}
SPL {X  -160.000, Y  +390.940, Z    +0.000, E1   +59.356, E3 +230553.628}
SPL {X  -159.620, Y  +374.678, Z    +0.000, E1   +59.299, E3 +230574.512}
SPL {X  -157.749, Y  +358.956, Z    +0.000, E1   +59.037, E3 +230596.210}
SPL {X  -154.809, Y  +345.275, Z    +0.000, E1   +58.527, E3 +230616.534}
SPL {X  -151.181, Y  +333.313, Z    +0.000, E1   +57.939, E3 +230635.242}
SPL {X  -146.730, Y  +321.901, Z    +0.000, E1   +57.169, E3 +230653.988}
SPL {X  -142.568, Y  +313.075, Z    +0.000, E1   +56.366, E3 +230669.109}
SPL {X  -139.172, Y  +306.763, Z    +0.000, E1   +55.717, E3 +230680.164}
SPL {X  -137.037, Y  +303.112, Z    +0.000, E1   +55.261, E3 +230686.711}
SPL {X  -123.439, Y  +283.902, Z    +0.000, E1   +48.158, E3 +230773.062}
ENDSPLINE

SPLINE
SPL {X  -141.803, Y  +311.593, Z    +0.000, E1   +37.608, E3 +230863.681}
SPL {X  -154.548, Y  +344.290, Z    +0.000, E1   +25.264, E3 +230888.164}
SPL {X  -159.249, Y  +370.212, Z    +0.000, E1   +11.801, E3 +230896.197}
SPL {X  -159.987, Y  +383.623, Z    +0.000, E1    +3.169, E3 +230897.950}
SPL {X  -160.000, Y  +388.238, Z    +0.000, E1    -0.420, E3 +230898.161}
SPL {X  -160.000, Y  +392.418, Z    +0.000, E1    -5.131, E3 +230898.401}
SPL {X  -160.000, Y  +399.157, Z    +0.000, E1   -14.351, E3 +230899.218}
SPL {X  -160.000, Y  +411.277, Z    +0.000, E1   -30.487, E3 +230901.996}
SPL {X  -160.000, Y  +452.990, Z    +0.000, E1   -53.470, E3 +230923.360}
SPL {X  -160.000, Y  +539.177, Z    +0.000, E1   -59.280, E3 +231001.686}
SPL {X  -160.000, Y  +554.731, Z    +0.000, E1   -59.281, E3 +231021.331}
SPL {X  -160.000, Y  +572.172, Z    +0.000, E1   -59.312, E3 +231043.294}
SPL {X  -160.000, Y  +589.502, Z    +0.000, E1   -59.284, E3 +231065.232}
SPL {X  -160.000, Y  +604.577, Z    +0.000, E1   -59.272, E3 +231084.291}
SPL {X  -160.000, Y  +620.386, Z    +0.000, E1   -59.294, E3 +231104.218}
SPL {X  -160.000, Y  +636.664, Z    +0.000, E1   -59.282, E3 +231124.808}
SPL {X  -160.000, Y  +654.257, Z    +0.000, E1   -59.312, E3 +231146.986}
SPL {X  -160.000, Y  +671.385, Z    +0.000, E1   -59.278, E3 +231168.675}
SPL {X  -159.497, Y  +687.081, Z    +0.000, E1   -59.218, E3 +231189.003}
SPL {X  -157.563, Y  +702.220, Z    +0.000, E1   -58.916, E3 +231210.164}
SPL {X  -154.922, Y  +714.390, Z    +0.000, E1   -58.446, E3 +231228.358}
SPL {X  -151.559, Y  +725.681, Z    +0.000, E1   -57.922, E3 +231245.988}
SPL {X  -147.777, Y  +735.736, Z    +0.000, E1   -57.226, E3 +231262.483}
SPL {X  -143.698, Y  +744.763, Z    +0.000, E1   -56.526, E3 +231277.759}
SPL {X  -138.992, Y  +753.654, Z    +0.000, E1   -55.630, E3 +231293.337}
SPL {X  -122.847, Y  +776.912, Z    +0.000, E1   -47.251, E3 +231403.019}
ENDSPLINE

SPLINE
SPL {X  -149.319, Y  +731.879, Z    +0.000, E1   -32.249, E3 +231497.406}
SPL {X  -158.304, Y  +697.637, Z    +0.000, E1   -16.440, E3 +231512.057}
SPL {X  -159.863, Y  +681.030, Z    +0.000, E1    -6.312, E3 +231514.999}
SPL {X  -160.000, Y  +673.530, Z    +0.000, E1    -1.059, E3 +231515.506}
SPL {X  -160.000, Y  +670.245, Z    +0.000, E1    +2.042, E3 +231515.619}
SPL {X  -160.000, Y  +663.790, Z    +0.000, E1   +10.467, E3 +231516.143}
SPL {X  -160.000, Y  +655.457, Z    +0.000, E1   +22.866, E3 +231517.506}
SPL {X  -160.000, Y  +644.540, Z    +0.000, E1   +36.054, E3 +231520.537}
SPL {X  -160.000, Y  +601.495, Z    +0.000, E1   +56.174, E3 +231541.466}
SPL {X  -160.000, Y  +515.545, Z    +0.000, E1   +60.629, E3 +231616.860}
SPL {X  -160.000, Y  +503.330, Z    +0.000, E1   +60.630, E3 +231631.466}
SPL {X  -160.000, Y  +487.139, Z    +0.000, E1   +60.676, E3 +231650.734}
SPL {X  -160.000, Y  +466.770, Z    +0.000, E1   +60.698, E3 +231675.029}
SPL {X  -160.000, Y  +454.269, Z    +0.000, E1   +59.898, E3 +231695.280}
ENDSPLINE

SPLINE
SPL {X  -160.000, Y  +458.973, Z    +0.000, E1   +55.880, E3 +231716.199}
ENDSPLINE

SPLINE
SPL {X  -160.000, Y  +435.816, Z    +0.000, E1   +57.237, E3 +231739.874}
SPL {X  -160.000, Y  +411.824, Z    +0.000, E1   +58.675, E3 +231762.368}
SPL {X  -160.000, Y  +390.940, Z    +0.000, E1   +59.356, E3 +231784.396}
SPL {X  -159.620, Y  +374.678, Z    +0.000, E1   +59.299, E3 +231805.280}
SPL {X  -157.749, Y  +358.956, Z    +0.000, E1   +59.037, E3 +231826.978}
SPL {X  -154.809, Y  +345.275, Z    +0.000, E1   +58.527, E3 +231847.301}
SPL {X  -151.181, Y  +333.313, Z    +0.000, E1   +57.939, E3 +231866.009}
SPL {X  -146.730, Y  +321.901, Z    +0.000, E1   +57.169, E3 +231884.755}
SPL {X  -142.568, Y  +313.075, Z    +0.000, E1   +56.366, E3 +231899.877}
SPL {X  -138.721, Y  +305.972, Z    +0.000, E1   +55.652, E3 +231912.305}
SPL {X  -123.439, Y  +283.902, Z    +0.000, E1   +48.158, E3 +232003.829}
ENDSPLINE

